(* AutoGeometry and AutoGroove-->Switch On/Off all Axis Power *)
	IF xToggleAllAxisPower THEN
		(* Step toggle Axis power *)
		CASE iStepAction OF
		(* check axis *)
		1:	IF NOT T_Station.TControl.xHardwareConfigError THEN
				xStepActionDone:=FALSE;
				iStepAction:=95;
				xTmp:=	T_Station.THardware.TAxisToolLeft.T_CtrleSingle.xDone
						AND T_Station.THardware.TAxisToolLeft.T_CtrleSingle.xNotMoving
						AND NOT(T_Station.THardware.TAxisToolLeft.T_CtrleSingle.xErr)
						AND NOT(T_Station.THardware.TAxisToolLeft.T_CtrleSingle.xExecute);
				xTmp:=	xTmp AND ((T_Station.THardware.TAxisToolCenter.T_CtrleSingle.xDone
						AND T_Station.THardware.TAxisToolCenter.T_CtrleSingle.xNotMoving
						AND NOT(T_Station.THardware.TAxisToolCenter.T_CtrleSingle.xErr)
						AND NOT(T_Station.THardware.TAxisToolCenter.T_CtrleSingle.xExecute) AND xMicroRodActive) OR NOT(xMicroRodActive)) ;
				xTmp:=	xTmp AND T_Station.THardware.TAxisToolRight.T_CtrleSingle.xDone
						AND T_Station.THardware.TAxisToolRight.T_CtrleSingle.xNotMoving
						AND NOT(T_Station.THardware.TAxisToolRight.T_CtrleSingle.xErr)
						AND NOT(T_Station.THardware.TAxisToolRight.T_CtrleSingle.xExecute);
				xTmp:=	xTmp AND T_Station.THardware.TAxisToolFeeder.T_CtrleSingle.xDone
						AND T_Station.THardware.TAxisToolFeeder.T_CtrleSingle.xNotMoving
						AND NOT(T_Station.THardware.TAxisToolFeeder.T_CtrleSingle.xErr)
						AND NOT(T_Station.THardware.TAxisToolFeeder.T_CtrleSingle.xExecute);
				xTmp:=	xTmp AND T_Station.THardware.TAxisGrindFeeder.T_CtrleSingle.xDone
						AND T_Station.THardware.TAxisGrindFeeder.T_CtrleSingle.xNotMoving
						AND NOT(T_Station.THardware.TAxisGrindFeeder.T_CtrleSingle.xErr)
						AND NOT(T_Station.THardware.TAxisGrindFeeder.T_CtrleSingle.xExecute);
				(* Start/Stop position or speed of teachin page has to be confirmed *)
				IF xTmp THEN
					iStepAction:=10;
				END_IF
			ELSE
				iStepAction:=95;
			END_IF;
		(* activ function axis *)
		10:	bStateMachine:=2;
			xSetStateMachine:=TRUE;
			xTmp:=	T_Station.THardware.TAxisToolLeft.T_CtrleSingle.xPower AND
					((T_Station.THardware.TAxisToolCenter.T_CtrleSingle.xPower AND xMicroRodActive) OR NOT(xMicroRodActive)) AND
					T_Station.THardware.TAxisToolRight.T_CtrleSingle.xPower AND
					T_Station.THardware.TAxisToolFeeder.T_CtrleSingle.xPower AND
					T_Station.THardware.TAxisGrindFeeder.T_CtrleSingle.xPower;
			IF xTmp THEN
				T_Station.THardware.TAxisToolLeft.T_CtrleSingle.iFunction:=4;
				IF xMicroRodActive THEN
					T_Station.THardware.TAxisToolCenter.T_CtrleSingle.iFunction:=4;
				END_IF;
				T_Station.THardware.TAxisToolRight.T_CtrleSingle.iFunction:=4;
				T_Station.THardware.TAxisToolFeeder.T_CtrleSingle.iFunction:=4;
				T_Station.THardware.TAxisGrindFeeder.T_CtrleSingle.iFunction:=4;
			ELSE
				IF NOT(T_Station.THardware.TAxisToolLeft.T_CtrleSingle.xPower) THEN
					T_Station.THardware.TAxisToolLeft.T_CtrleSingle.iFunction:=3;
				END_IF;
				IF xMicroRodActive THEN
					IF NOT(T_Station.THardware.TAxisToolCenter.T_CtrleSingle.xPower) THEN
						T_Station.THardware.TAxisToolCenter.T_CtrleSingle.iFunction:=3;
					END_IF;
				END_IF;
				IF NOT(T_Station.THardware.TAxisToolRight.T_CtrleSingle.xPower) THEN
					T_Station.THardware.TAxisToolRight.T_CtrleSingle.iFunction:=3;
				END_IF;
				IF NOT(T_Station.THardware.TAxisToolFeeder.T_CtrleSingle.xPower) THEN
					T_Station.THardware.TAxisToolFeeder.T_CtrleSingle.iFunction:=3;
				END_IF;
				IF NOT(T_Station.THardware.TAxisGrindFeeder.T_CtrleSingle.xPower) THEN
					T_Station.THardware.TAxisGrindFeeder.T_CtrleSingle.iFunction:=3;
				END_IF;
			END_IF;
			T_Station.THardware.TAxisToolLeft.T_CtrleSingle.xExecute:=TRUE;
			T_Station.THardware.TAxisToolCenter.T_CtrleSingle.xExecute:=xMicroRodActive;
			T_Station.THardware.TAxisToolRight.T_CtrleSingle.xExecute:=TRUE;
			T_Station.THardware.TAxisToolFeeder.T_CtrleSingle.xExecute:=TRUE;
			T_Station.THardware.TAxisGrindFeeder.T_CtrleSingle.xExecute:=TRUE;
			(* next step *)
			iStepAction:=20;
			xStepActionDone:=FALSE;
		(* confirm execution *)
		20:	IF NOT(xStepActionDone) THEN
			(* confirm execution *)
				T_Station.THardware.TAxisToolLeft.T_CtrleSingle.xExecute:=FALSE;
				T_Station.THardware.TAxisToolCenter.T_CtrleSingle.xExecute:=FALSE;
				T_Station.THardware.TAxisToolRight.T_CtrleSingle.xExecute:=FALSE;
				T_Station.THardware.TAxisToolFeeder.T_CtrleSingle.xExecute:=FALSE;
				T_Station.THardware.TAxisGrindFeeder.T_CtrleSingle.xExecute:=FALSE;
				xStepActionDone:=TRUE;
			ELSE
				xTmp:=	T_Station.THardware.TAxisToolLeft.T_CtrleSingle.xDone AND
						((T_Station.THardware.TAxisToolCenter.T_CtrleSingle.xDone AND xMicroRodActive) OR NOT(xMicroRodActive)) AND
						T_Station.THardware.TAxisToolRight.T_CtrleSingle.xDone AND
						T_Station.THardware.TAxisToolFeeder.T_CtrleSingle.xDone AND
						T_Station.THardware.TAxisGrindFeeder.T_CtrleSingle.xDone;
				IF xTmp THEN
				(* confirm action next step *)
					bStateMachine:=1;
					xSetStateMachine:=TRUE;
					iStepAction:=90;
					xStepActionDone:=FALSE;
				ELSE
					xTmp:=	T_Station.THardware.TAxisToolLeft.T_CtrleSingle.xErr OR
							(T_Station.THardware.TAxisToolCenter.T_CtrleSingle.xErr AND xMicroRodActive) OR
							T_Station.THardware.TAxisToolRight.T_CtrleSingle.xErr OR
							T_Station.THardware.TAxisToolFeeder.T_CtrleSingle.xErr OR
							T_Station.THardware.TAxisGrindFeeder.T_CtrleSingle.xErr;
					IF xTmp THEN
					(* activ action not ready or error *)
						iStepAction:=99;
						xStepActionDone:=FALSE;
					END_IF
				END_IF
			END_IF
		(* action done *)
		90:	T_Visu.ptrT_ExchgParam^.T_StationCommon.wState:=T_Visu.ptrT_ExchgParam^.T_StationCommon.wState AND 16#BF;
			T_Visu.T_CtrleAction.xDone:=TRUE;
			T_Visu.T_CtrleAction.xNotReady:=FALSE;
			T_Visu.T_CtrleAction.xErr:=FALSE;
			T_Visu.T_CtrleAction.udiErrorID:=0;
			xToggleAllAxisPower:=FALSE;
		(* axis not ready *)
		95:	T_Visu.ptrT_ExchgParam^.T_StationCommon.wState:=T_Visu.ptrT_ExchgParam^.T_StationCommon.wState AND 16#BF;
			TimerNotReady(IN:=TRUE);
			xToggleAllAxisPower:=FALSE;
		(* error *)
		99:	T_Visu.ptrT_ExchgParam^.T_StationCommon.wState:=T_Visu.ptrT_ExchgParam^.T_StationCommon.wState AND 16#BF;
			T_Visu.T_CtrleAction.xDone:=TRUE;
			T_Visu.T_CtrleAction.xNotReady:=FALSE;
			diErrorNr:=0;
			IF T_Station.THardware.TAxisToolLeft.T_CtrleSingle.xErr THEN
				diErrorNr:=1000000 + T_Station.THardware.TAxisToolLeft.T_CtrleSingle.udiErrorID;
			END_IF;
			IF xMicroRodActive THEN
				IF T_Station.THardware.TAxisToolCenter.T_CtrleSingle.xErr THEN
					diErrorNr:=2000000 + T_Station.THardware.TAxisToolCenter.T_CtrleSingle.udiErrorID;
				END_IF;
			END_IF;
			IF T_Station.THardware.TAxisToolRight.T_CtrleSingle.xErr THEN
				diErrorNr:=3000000 + T_Station.THardware.TAxisToolRight.T_CtrleSingle.udiErrorID;
			END_IF;
			IF T_Station.THardware.TAxisToolFeeder.T_CtrleSingle.xErr THEN
				diErrorNr:=4000000 + T_Station.THardware.TAxisToolFeeder.T_CtrleSingle.udiErrorID;
			END_IF;
			IF T_Station.THardware.TAxisGrindFeeder.T_CtrleSingle.xErr THEN
				diErrorNr:=5000000 + T_Station.THardware.TAxisGrindFeeder.T_CtrleSingle.udiErrorID;
			END_IF;
			FBErrorMessage(	diErrorNr:=diErrorNr,
							T_ErrorList:=T_ErrorList);
			T_Visu.ptrT_ExchgParam^.T_Visu.T_Message.sDynamicTextEnglish:=FBErrorMessage.sErrorTextEnglish;
			T_Visu.ptrT_ExchgParam^.T_Visu.T_Message.sDynamicTextDeutsch:=FBErrorMessage.sErrorTextDeutsch;
			T_Visu.ptrT_ExchgParam^.T_Visu.T_Message.sDynamicTextFrancais:=FBErrorMessage.sErrorTextFrancais;
			T_Visu.ptrT_ExchgParam^.T_SafetyCtrl.xSetForceError:=TRUE;
			T_Visu.ptrT_ExchgParam^.T_SafetyCtrl.diSetForceErrorNr:=diErrorNr;
			T_Visu.T_CtrleAction.xErr:=FALSE;
			T_Visu.T_CtrleAction.udiErrorID:=0;
			T_Station.THardware.TAxisToolLeft.T_CtrleSingle.iFunction:=1;
			T_Station.THardware.TAxisToolLeft.T_CtrleSingle.xExecute:=T_Station.THardware.TAxisToolLeft.T_CtrleSingle.xErr;
			IF xMicroRodActive THEN
				T_Station.THardware.TAxisToolCenter.T_CtrleSingle.iFunction:=1;
				T_Station.THardware.TAxisToolCenter.T_CtrleSingle.xExecute:=T_Station.THardware.TAxisToolCenter.T_CtrleSingle.xErr;
			END_IF;
			T_Station.THardware.TAxisToolRight.T_CtrleSingle.iFunction:=1;
			T_Station.THardware.TAxisToolRight.T_CtrleSingle.xExecute:=T_Station.THardware.TAxisToolRight.T_CtrleSingle.xErr;
			T_Station.THardware.TAxisToolFeeder.T_CtrleSingle.iFunction:=1;
			T_Station.THardware.TAxisToolFeeder.T_CtrleSingle.xExecute:=T_Station.THardware.TAxisToolFeeder.T_CtrleSingle.xErr;
			T_Station.THardware.TAxisGrindFeeder.T_CtrleSingle.iFunction:=1;
			T_Station.THardware.TAxisGrindFeeder.T_CtrleSingle.xExecute:=T_Station.THardware.TAxisGrindFeeder.T_CtrleSingle.xErr;
			xToggleAllAxisPower:=FALSE;
		END_CASE
	END_IF

(* Correction Tool Diameter +,++,-,-- *)
	IF xCorrectionToolDiameterAdd OR xCorrectionToolDiameterAddMore OR 	xCorrectionToolDiameterSub OR xCorrectionToolDiameterSubMore OR xResetToolDiameterCorrection OR xKeyPadActivation THEN
		CASE iStepAction OF
		(* check visu *)
		1:	xTmp:=	TRUE;
			IF xTmp THEN
				(* next Step *)
				iStepAction :=10;
				IF xResetToolDiameterCorrection THEN
					(* next Step *)
					iStepAction :=20;
				END_IF;
				IF xKeyPadActivation THEN
					IF (T_Visu.T_PlcParam.dwActualPage = 420) OR (T_Visu.T_PlcParam.dwActualPage = 11) OR (T_Visu.T_PlcParam.dwActualPage = 21) THEN
						(* next Step *)
						iStepAction :=30;
					END_IF;
					IF (T_Visu.T_PlcParam.dwActualPage = 430) THEN
						(* next Step *)
						iStepAction :=40;
					END_IF;
				END_IF;
			(* activ error *)
			ELSE iStepAction:=95; END_IF
		10:	IF xCorrectionToolDiameterAdd THEN
				rCorrectionValue:=0.1;
			END_IF;
			IF xCorrectionToolDiameterAddMore THEN
				rCorrectionValue:=1.0;
			END_IF;
			IF xCorrectionToolDiameterSub THEN
				rCorrectionValue:=-0.1;
			END_IF;
			IF xCorrectionToolDiameterSubMore THEN
				rCorrectionValue:=-1.0;
			END_IF;
			T_Visu.ptrT_ExchgParam^.T_InfoValueCommon.rCorrectionToolDiameter:=T_Visu.ptrT_ExchgParam^.T_InfoValueCommon.rCorrectionToolDiameter + rCorrectionValue;
			IF (T_Visu.ptrT_ExchgParam^.T_InfoValueCommon.rCorrectionToolDiameter < 0.1) AND
			    (T_Visu.ptrT_ExchgParam^.T_InfoValueCommon.rCorrectionToolDiameter > -0.1) THEN
				T_Visu.ptrT_ExchgParam^.T_InfoValueCommon.rCorrectionToolDiameter:=0.0;
			END_IF;
			(* next Step *)
			iStepAction :=90;
		20:	T_Visu.ptrT_ExchgParam^.T_InfoValueCommon.rCorrectionToolDiameter:=0.0;
			(* next Step *)
			iStepAction :=90;
		30:	T_Visu.ptrT_ExchgParam^.T_InfoValueCommon.xKeyPadActivation:=NOT(T_Visu.ptrT_ExchgParam^.T_InfoValueCommon.xKeyPadActivation);
			(* next Step *)
			iStepAction :=90;
		40:	(* 0= 3 value prisma, 1 = 3 value prisma input para, 2 = 2 value prisma, 3 = 2 value prisma input para *)
			IF (T_Visu.ptrT_ExchgParam^.T_StationCommon.T_PrismPara.bStateInputPrisma = 0) THEN
				T_Visu.ptrT_ExchgParam^.T_StationCommon.T_PrismPara.bStateInputPrisma:=1;
			ELSIF (T_Visu.ptrT_ExchgParam^.T_StationCommon.T_PrismPara.bStateInputPrisma = 1) THEN
				T_Visu.ptrT_ExchgParam^.T_StationCommon.T_PrismPara.bStateInputPrisma:=0;
			ELSIF (T_Visu.ptrT_ExchgParam^.T_StationCommon.T_PrismPara.bStateInputPrisma = 2) THEN
				T_Visu.ptrT_ExchgParam^.T_StationCommon.T_PrismPara.bStateInputPrisma:=3;
			ELSIF (T_Visu.ptrT_ExchgParam^.T_StationCommon.T_PrismPara.bStateInputPrisma = 3) THEN
				T_Visu.ptrT_ExchgParam^.T_StationCommon.T_PrismPara.bStateInputPrisma:=2;
			END_IF;
			(* next Step *)
			iStepAction:=90;
		(* change page done *)
		90:	T_Visu.T_CtrleAction.xDone:=TRUE;
			T_Visu.T_CtrleAction.xNotReady:=FALSE;
			T_Visu.T_CtrleAction.xErr:=FALSE;
			T_Visu.T_CtrleAction.udiErrorID:=0;
			xCorrectionToolDiameterAdd:=xCorrectionToolDiameterAddMore:=xCorrectionToolDiameterSub:=xCorrectionToolDiameterSubMore:=xResetToolDiameterCorrection:=xKeyPadActivation:=FALSE;
		(* not ready *)
		95:	T_Visu.T_CtrleAction.xDone:=TRUE;
			T_Visu.T_CtrleAction.xNotReady:=FALSE;
			T_Visu.T_CtrleAction.xErr:=FALSE;
			T_Visu.T_CtrleAction.udiErrorID:=0;
			xCorrectionToolDiameterAdd:=xCorrectionToolDiameterAddMore:=xCorrectionToolDiameterSub:=xCorrectionToolDiameterSubMore:=xResetToolDiameterCorrection:=xKeyPadActivation:=FALSE;
		END_CASE
	END_IF;

(* Function Correction Tool Diameter *)
	IF xFctCorrectionToolDiameter THEN
		CASE iStepAction OF
		(* check axis *)
		1:	IF NOT T_Station.TControl.xHardwareConfigError THEN
				xStepActionDone:=FALSE;
				iStepAction:=95;
				xTmp:=	T_Station.THardware.TAxisGrindFeeder.T_CtrleSingle.xDone
						AND T_Station.THardware.TAxisGrindFeeder.T_CtrleSingle.xReady
						AND T_Station.THardware.TAxisGrindFeeder.T_CtrleSingle.xNotMoving
						AND NOT(T_Station.THardware.TAxisGrindFeeder.T_CtrleSingle.xErr)
						AND NOT(T_Station.THardware.TAxisGrindFeeder.T_CtrleSingle.xExecute);
				(* Start/Stop position or speed of teachin page has to be confirmed *)
				IF xTmp THEN
					iStepAction:=10;
				END_IF
			ELSE
				iStepAction:=95;
			END_IF;
		(* Display message to ask for confirmation *)
		10:	T_Visu.ptrT_ExchgParam^.T_Visu.T_Message.iState:=108;
			iStepAction:=20;
		(* waiting for key <Enter> or <Esc> *)
		20:	IF RisingEdgeKeyPanel_Enter.Q THEN iStepAction:=30;
			ELSE IF RisingEdgeKeyPanel_Esc.Q THEN iStepAction:=90; END_IF END_IF
			(* An other message has been displayed, stop teach action *)
			IF T_Visu.ptrT_ExchgParam^.T_Visu.T_Message.iState<>108 THEN iStepAction:=90; END_IF
		(* activ function axis *)
		30:	(*T_Visu.ptrT_ExchgParam^.T_InfoValueCommon.rActualGrindAxisPosition:=T_Visu.ptrT_ExchgParam^.T_InfoValueCommon.rActualGrindAxisPosition - T_Visu.ptrT_ExchgParam^.T_InfoValueCommon.rCorrectionToolDiameter;*)
			T_Station.THardware.TAxisGrindFeeder.T_CtrleSingle.rSetPosition:=T_Station.THardware.TAxisGrindFeeder.T_LiveValue.lrActualPosition - T_Visu.ptrT_ExchgParam^.T_InfoValueCommon.rCorrectionToolDiameter;
			T_Visu.ptrT_ExchgParam^.T_InfoValueCommon.rCorrectionToolDiameter:=0.0;
			T_Station.THardware.TAxisGrindFeeder.T_CtrleSingle.iFunction:=11;
			T_Station.THardware.TAxisGrindFeeder.T_CtrleSingle.xExecute:=TRUE;
			(* next step *)
			iStepAction:=50;
			xStepActionDone:=FALSE;
		(* confirm execution *)
		50:	IF NOT(xStepActionDone) THEN
			(* confirm execution *)
				T_Station.THardware.TAxisGrindFeeder.T_CtrleSingle.xExecute:=FALSE;
				xStepActionDone:=TRUE;
			ELSE
				IF T_Station.THardware.TAxisGrindFeeder.T_CtrleSingle.xDone THEN
				(* confirm action next step *)
					iStepAction:=90;
					xStepActionDone:=FALSE;
				ELSE
					IF T_Station.THardware.TAxisGrindFeeder.T_CtrleSingle.xErr THEN
					(* activ action not ready or error *)
						iStepAction:=99;
						xStepActionDone:=FALSE;
					END_IF
				END_IF
			END_IF
		(* action done *)
		90:	T_Visu.ptrT_ExchgParam^.T_StationCommon.wState:=T_Visu.ptrT_ExchgParam^.T_StationCommon.wState AND 16#BF;
			T_Visu.T_CtrleAction.xDone:=TRUE;
			T_Visu.T_CtrleAction.xNotReady:=FALSE;
			T_Visu.T_CtrleAction.xErr:=FALSE;
			T_Visu.T_CtrleAction.udiErrorID:=0;
			xFctCorrectionToolDiameter:=FALSE;
		(* axis not ready *)
		95:	T_Visu.ptrT_ExchgParam^.T_StationCommon.wState:=T_Visu.ptrT_ExchgParam^.T_StationCommon.wState AND 16#BF;
			TimerNotReady(IN:=TRUE);
			xFctCorrectionToolDiameter:=FALSE;
		(* error *)
		99:	T_Visu.ptrT_ExchgParam^.T_StationCommon.wState:=T_Visu.ptrT_ExchgParam^.T_StationCommon.wState AND 16#BF;
			T_Visu.T_CtrleAction.xDone:=TRUE;
			T_Visu.T_CtrleAction.xNotReady:=FALSE;
			IF (T_Station.THardware.TAxisGrindFeeder.T_Config_Gen.iTyp <> 0) THEN
				diErrorNr:=(T_Station.THardware.TAxisGrindFeeder.T_Config_Gen.iTyp * 1000000) + T_Station.THardware.TAxisGrindFeeder.T_CtrleSingle.udiErrorID;
			ELSE
				diErrorNr:=0;
			END_IF;
			FBErrorMessage(	diErrorNr:=diErrorNr,
							T_ErrorList:=T_ErrorList);
			T_Visu.ptrT_ExchgParam^.T_Visu.T_Message.sDynamicTextEnglish:=FBErrorMessage.sErrorTextEnglish;
			T_Visu.ptrT_ExchgParam^.T_Visu.T_Message.sDynamicTextDeutsch:=FBErrorMessage.sErrorTextDeutsch;
			T_Visu.ptrT_ExchgParam^.T_Visu.T_Message.sDynamicTextFrancais:=FBErrorMessage.sErrorTextFrancais;
			T_Visu.ptrT_ExchgParam^.T_SafetyCtrl.xSetForceError:=TRUE;
			T_Visu.ptrT_ExchgParam^.T_SafetyCtrl.diSetForceErrorNr:=diErrorNr;
			T_Visu.T_CtrleAction.xErr:=FALSE;
			T_Visu.T_CtrleAction.udiErrorID:=0;
			T_Station.THardware.TAxisGrindFeeder.T_CtrleSingle.iFunction:=1;
			T_Station.THardware.TAxisGrindFeeder.T_CtrleSingle.xExecute:=TRUE;
			xFctCorrectionToolDiameter:=FALSE;
		END_CASE
	END_IF;

(* Select Prisma 1 or 2 Input *)
	IF xSelectPrisma THEN
		CASE iStepAction OF
		(* check visu *)
		1:	xTmp:=	TRUE;
			IF xTmp THEN
				(* next Step *)
				iStepAction :=10;
			(* activ error *)
			ELSE iStepAction:=95; END_IF
		10:	(* 0= 3 value prisma, 1 = 3 value prisma input para, 2 = 2 value prisma, 3 = 2 value prisma input para *)
			IF (T_Visu.ptrT_ExchgParam^.T_StationCommon.T_PrismPara.bStateInputPrisma = 0) OR (T_Visu.ptrT_ExchgParam^.T_StationCommon.T_PrismPara.bStateInputPrisma = 1) THEN
				T_Visu.ptrT_ExchgParam^.T_StationCommon.T_PrismPara.bStateInputPrisma:=2;
			ELSIF (T_Visu.ptrT_ExchgParam^.T_StationCommon.T_PrismPara.bStateInputPrisma = 2) OR (T_Visu.ptrT_ExchgParam^.T_StationCommon.T_PrismPara.bStateInputPrisma = 3) THEN
				T_Visu.ptrT_ExchgParam^.T_StationCommon.T_PrismPara.bStateInputPrisma:=0;
			END_IF;
			(* next Step *)
			iStepAction:=90;
		(* change page done *)
		90:	T_Visu.T_CtrleAction.xDone:=TRUE;
			T_Visu.T_CtrleAction.xNotReady:=FALSE;
			T_Visu.T_CtrleAction.xErr:=FALSE;
			T_Visu.T_CtrleAction.udiErrorID:=0;
			xSelectPrisma:=FALSE;
		(* not ready *)
		95:	T_Visu.T_CtrleAction.xDone:=TRUE;
			T_Visu.T_CtrleAction.xNotReady:=FALSE;
			T_Visu.T_CtrleAction.xErr:=FALSE;
			T_Visu.T_CtrleAction.udiErrorID:=0;
			xSelectPrisma:=FALSE;
		END_CASE
	END_IF;

(* Set calculated ToolRotation Torque *)
	IF xSetCalculToolRotTorque THEN
		CASE iStepAction OF
		(* check visu *)
		1:	xTmp:=	TRUE;
			IF xTmp THEN
				(* next Step *)
				iStepAction :=10;
			(* activ error *)
			ELSE iStepAction:=95; END_IF
		10:	uiToolLeftZeroTorque:=T_Station.THardware.TAxisToolLeft.T_LiveValue.uiActualTorque;
			FBCalcTorqueToolLeft(	xStart:=TRUE,
									uiActualTorque:= T_Station.THardware.TAxisToolLeft.T_LiveValue.uiActualTorque,
									uiZeroTorque:=uiToolLeftZeroTorque,
									iStepCalc:= 100);
			uiToolCenterZeroTorque:=T_Station.THardware.TAxisToolCenter.T_LiveValue.uiActualTorque;
			FBCalcTorqueToolCenter(	xStart:=TRUE,
									uiActualTorque:= T_Station.THardware.TAxisToolCenter.T_LiveValue.uiActualTorque,
									uiZeroTorque:=uiToolCenterZeroTorque,
									iStepCalc:= 100);
			uiToolRightZeroTorque:=T_Station.THardware.TAxisToolRight.T_LiveValue.uiActualTorque;
			FBCalcTorqueToolRight(	xStart:=TRUE,
									uiActualTorque:= T_Station.THardware.TAxisToolRight.T_LiveValue.uiActualTorque,
									uiZeroTorque:=uiToolRightZeroTorque,
									iStepCalc:= 100);
			(* next Step *)
			iStepAction:=90;
		(* change page done *)
		90:	T_Visu.T_CtrleAction.xDone:=TRUE;
			T_Visu.T_CtrleAction.xNotReady:=FALSE;
			T_Visu.T_CtrleAction.xErr:=FALSE;
			T_Visu.T_CtrleAction.udiErrorID:=0;
			xSetCalculToolRotTorque:=FALSE;
		(* not ready *)
		95:	T_Visu.T_CtrleAction.xDone:=TRUE;
			T_Visu.T_CtrleAction.xNotReady:=FALSE;
			T_Visu.T_CtrleAction.xErr:=FALSE;
			T_Visu.T_CtrleAction.udiErrorID:=0;
			xSetCalculToolRotTorque:=FALSE;
		END_CASE
	END_IF;

(* Reset calculated ToolRotation Torque *)
	IF xResetCalculToolRotTorque THEN
		CASE iStepAction OF
		(* check visu *)
		1:	xTmp:=	TRUE;
			IF xTmp THEN
				(* next Step *)
				iStepAction :=10;
			(* activ error *)
			ELSE iStepAction:=95; END_IF
		10:	uiToolLeftZeroTorque:=0;
			FBCalcTorqueToolLeft(	xStart:=TRUE,
									uiActualTorque:= T_Station.THardware.TAxisToolLeft.T_LiveValue.uiActualTorque,
									uiZeroTorque:=uiToolLeftZeroTorque,
									iStepCalc:= 100);
			uiToolCenterZeroTorque:=0;
			FBCalcTorqueToolCenter(	xStart:=TRUE,
									uiActualTorque:= T_Station.THardware.TAxisToolCenter.T_LiveValue.uiActualTorque,
									uiZeroTorque:=uiToolCenterZeroTorque,
									iStepCalc:= 100);
			uiToolRightZeroTorque:=0;
			FBCalcTorqueToolRight(	xStart:=TRUE,
									uiActualTorque:= T_Station.THardware.TAxisToolRight.T_LiveValue.uiActualTorque,
									uiZeroTorque:=uiToolRightZeroTorque,
									iStepCalc:= 100);
			(* next Step *)
			iStepAction:=90;
		(* change page done *)
		90:	T_Visu.T_CtrleAction.xDone:=TRUE;
			T_Visu.T_CtrleAction.xNotReady:=FALSE;
			T_Visu.T_CtrleAction.xErr:=FALSE;
			T_Visu.T_CtrleAction.udiErrorID:=0;
			xResetCalculToolRotTorque:=FALSE;
		(* not ready *)
		95:	T_Visu.T_CtrleAction.xDone:=TRUE;
			T_Visu.T_CtrleAction.xNotReady:=FALSE;
			T_Visu.T_CtrleAction.xErr:=FALSE;
			T_Visu.T_CtrleAction.udiErrorID:=0;
			xResetCalculToolRotTorque:=FALSE;
		END_CASE
	END_IF;

(* Switch WireFeed Jog Speed Slow/Fast *)
	IF xSlowFastJogToolRotation OR xSlowFastJogToolFeeder OR xSlowFastJogGrindFeeder THEN
		CASE iStepAction OF
		(* check visu *)
		1:	xTmp:=	TRUE;
			IF xTmp THEN
				(* next Step *)
				iStepAction :=10;
			(* activ error *)
			ELSE iStepAction:=95; END_IF
		10:	IF xSlowFastJogToolRotation THEN
				T_Visu.ptrT_ExchgParam^.T_TeachIn.xSlowFastToolRotation:=NOT(T_Visu.ptrT_ExchgParam^.T_TeachIn.xSlowFastToolRotation);
			END_IF;
			IF xSlowFastJogToolFeeder THEN
				T_Visu.ptrT_ExchgParam^.T_TeachIn.xSlowFastToolFeed:=NOT(T_Visu.ptrT_ExchgParam^.T_TeachIn.xSlowFastToolFeed);
			END_IF;
			IF xSlowFastJogGrindFeeder THEN
				T_Visu.ptrT_ExchgParam^.T_TeachIn.xSlowFastGrindFeeder:=NOT(T_Visu.ptrT_ExchgParam^.T_TeachIn.xSlowFastGrindFeeder);
			END_IF;
			(* next Step *)
			iStepAction:=90;
		(* change page done *)
		90:	T_Visu.T_CtrleAction.xDone:=TRUE;
			T_Visu.T_CtrleAction.xNotReady:=FALSE;
			T_Visu.T_CtrleAction.xErr:=FALSE;
			T_Visu.T_CtrleAction.udiErrorID:=0;
			xSlowFastJogToolRotation:=xSlowFastJogToolFeeder:=xSlowFastJogGrindFeeder:=FALSE;
		(* not ready *)
		95:	T_Visu.T_CtrleAction.xDone:=TRUE;
			T_Visu.T_CtrleAction.xNotReady:=FALSE;
			T_Visu.T_CtrleAction.xErr:=FALSE;
			T_Visu.T_CtrleAction.udiErrorID:=0;
			xSlowFastJogToolRotation:=xSlowFastJogToolFeeder:=xSlowFastJogGrindFeeder:=FALSE;
		END_CASE
	END_IF;

(* Action stop axis *)
	IF xStopAxis THEN
		(* Step stop axis *)
		CASE iStepAction OF
		(* check axis *)
		1:	xMoveAbsPosition:=xMoveRelPosition:=xMoveContinousVel:=FALSE;
			IF NOT T_Station.TControl.xHardwareConfigError THEN
				xStepActionDone:=FALSE;
				IF ptrTeachINAxis^.T_CtrleSingle.xErr THEN
					iStepAction:=99;
					RETURN;
				END_IF;
				iStepAction:=95;
				xTmp:=	ptrTeachINAxis^.T_CtrleSingle.xReady (*AND
						NOT(ptrTeachINAxis^.T_CtrleSingle.xErr)*);
				(* Start/Stop position or speed of teachin page has to be confirmed *)
				IF xTmp THEN
					iStepAction:=10;
				ELSE
					iStepAction:=95;
				END_IF
			ELSE
				iStepAction:=95;
			END_IF;
		(* activ function axis *)
		10:	ptrTeachINAxis^.T_CtrleSingle.iFunction:=5;
			ptrTeachINAxis^.T_CtrleSingle.xExecute:=TRUE;
			(* init. acc/dec/jerk *)
			ptrTeachINAxis^.T_CtrleSingle.lrAcceleration:=TParaAxisTeachIN.rAcceleration;
			ptrTeachINAxis^.T_CtrleSingle.lrDecceleration:=TParaAxisTeachIN.rDeceleration;
			(*
			ptrTeachINAxis^.T_CtrleSingle.lrAcceleration:=ptrTeachINAxis^.T_Config_ObjFileValue.lrAcceleration;
			ptrTeachINAxis^.T_CtrleSingle.lrDecceleration:=ptrTeachINAxis^.T_Config_ObjFileValue.lrDecceleration;
			ptrTeachINAxis^.T_CtrleSingle.lrJerk:=ptrTeachINAxis^.T_Config_ObjFileValue.lrJerk;
			*)
			(* next step *)
			iStepAction:=20;
			xStepActionDone:=FALSE;
		(* waiting stop confirmation *)
		20:	IF NOT(xStepActionDone) THEN
			(* confirm execution *)
				ptrTeachINAxis^.T_CtrleSingle.xExecute:=FALSE;
				xStepActionDone:=TRUE;
			ELSE
				IF ptrTeachINAxis^.T_CtrleSingle.xDone THEN
				(* confirm action next step *)
					iStepAction:=90;
					xStepActionDone:=FALSE;
				ELSE
					IF ptrTeachINAxis^.T_CtrleSingle.xErr THEN
					(* activ action not ready or error *)
						iStepAction:=99;
						xStepActionDone:=FALSE;
					END_IF
				END_IF
			END_IF
		(* waiting time out *)
		89:	IF TimerAction.Q THEN iStepAction:=90; END_IF
			(*T_Visu.ptrT_ExchgParam^.T_TeachIn.iStateAxisMovement:=1;*)
		(* action done *)
		90:	bStateMachine:=1;
			xSetStateMachine:=TRUE;
			T_Visu.ptrT_ExchgParam^.T_StationCommon.wState:=T_Visu.ptrT_ExchgParam^.T_StationCommon.wState AND 16#BF;
			T_Visu.T_CtrleAction.xDone:=TRUE;
			T_Visu.T_CtrleAction.xNotReady:=FALSE;
			T_Visu.T_CtrleAction.xErr:=FALSE;
			T_Visu.T_CtrleAction.udiErrorID:=0;
			xStopAxis:=FALSE;
			(*T_Visu.ptrT_ExchgParam^.T_TeachIn.iStateAxisMovement:=1;*)
		(* axis not ready *)
		95:	T_Visu.ptrT_ExchgParam^.T_StationCommon.wState:=T_Visu.ptrT_ExchgParam^.T_StationCommon.wState AND 16#BF;
			TimerNotReady(IN:=TRUE);
			xStopAxis:=FALSE;
			(*T_Visu.ptrT_ExchgParam^.T_TeachIn.iStateAxisMovement:=1;*)
		(* error *)
		99:	T_Visu.ptrT_ExchgParam^.T_StationCommon.wState:=T_Visu.ptrT_ExchgParam^.T_StationCommon.wState AND 16#BF;
			T_Visu.T_CtrleAction.xDone:=TRUE;
			T_Visu.T_CtrleAction.xNotReady:=FALSE;
			IF (ptrTeachINAxis^.T_Config_Gen.iTyp <> 0) THEN
				diErrorNr:=(ptrTeachINAxis^.T_Config_Gen.iTyp * 1000000) + ptrTeachINAxis^.T_CtrleSingle.udiErrorID;
			ELSE
				diErrorNr:=0;
			END_IF;
			FBErrorMessage(	diErrorNr:=diErrorNr,
							T_ErrorList:=T_ErrorList);
			T_Visu.ptrT_ExchgParam^.T_Visu.T_Message.sDynamicTextEnglish:=FBErrorMessage.sErrorTextEnglish;
			T_Visu.ptrT_ExchgParam^.T_Visu.T_Message.sDynamicTextDeutsch:=FBErrorMessage.sErrorTextDeutsch;
			T_Visu.ptrT_ExchgParam^.T_Visu.T_Message.sDynamicTextFrancais:=FBErrorMessage.sErrorTextFrancais;
			T_Visu.ptrT_ExchgParam^.T_SafetyCtrl.xSetForceError:=TRUE;
			T_Visu.ptrT_ExchgParam^.T_SafetyCtrl.diSetForceErrorNr:=diErrorNr;
			T_Visu.T_CtrleAction.xErr:=FALSE;
			T_Visu.T_CtrleAction.udiErrorID:=0;
			ptrTeachINAxis^.T_CtrleSingle.iFunction:=1;
			ptrTeachINAxis^.T_CtrleSingle.xExecute:=TRUE;
			xStopAxis:=FALSE;
			T_StartUp.T_Ctrle.xSetSecurityStateON:=TRUE;
		END_CASE
	END_IF

(* Action move abs position *)
	IF xMoveAbsPosition OR xMoveRelPosition THEN
		(* Step move abs position *)
		CASE iStepAction OF
		(* check axis *)
		1:	IF NOT T_Station.TControl.xHardwareConfigError THEN
				xStepActionDone:=FALSE;
				iStepAction:=95;
				xTmp:=	ptrTeachINAxis^.T_CtrleSingle.xDone
						AND ptrTeachINAxis^.T_CtrleSingle.xReady
						AND ptrTeachINAxis^.T_CtrleSingle.xNotMoving
						AND ptrTeachINAxis^.T_CtrleSingle.xPower
						AND NOT(ptrTeachINAxis^.T_CtrleSingle.xErr)
						AND NOT(ptrTeachINAxis^.T_CtrleSingle.xExecute)
(*24.09.2010: KFS	{	 *)
						AND( (  T_Visu.T_PlcParam.dwActualPage = 210
							   AND NOT(T_Station.THardware.TCylToolLeftActive.T_CtrleCyl.T_Standard.xActivOn)
							   AND NOT(T_Station.THardware.TCylToolRightActive.T_CtrleCyl.T_Standard.xActivOn)
					     		   AND NOT(T_Station.THardware.TCylToolCenterActive.T_CtrleCyl.T_Standard.xActivOn) )  OR ( T_Visu.T_PlcParam.dwActualPage <> 210))
(*24.09.2010: KFS	}	 *)
						AND ((ptrTeachINAxis^.T_CtrleSingle.xRef AND xMoveAbsPosition AND xMicroRodActive) OR NOT(xMicroRodActive)OR xMoveRelPosition);
				(* Start/Stop position or speed of teachin page has to be confirmed *)
				IF xTmp THEN
					iStepAction:=10;
				ELSE
					IF NOT ptrTeachINAxis^.T_CtrleSingle.xRef AND xMoveAbsPosition THEN
					(* Display message, axis not referenced *)
						tTimeOutAction:=TimerAction.ET+T#2s;
						T_Visu.ptrT_ExchgParam^.T_Visu.T_Message.iState:=18;
						(* Action has been cancelled *)
						iStepAction:=89;
					END_IF
				END_IF
			ELSE
				iStepAction:=95;
			END_IF;
		(* activ function axis *)
		10:	tTimeOutAction:=T#999s;
			bStateMachine:=2;
			xSetStateMachine:=TRUE;
			IF xMoveAbsPosition THEN iStepAction:=20; END_IF
			IF xMoveRelPosition THEN iStepAction:=35; END_IF
			(* init. acc/dec/jerk *)
			ptrTeachINAxis^.T_CtrleSingle.lrAcceleration:=TParaAxisTeachIN.rAcceleration;
			ptrTeachINAxis^.T_CtrleSingle.lrDecceleration:=TParaAxisTeachIN.rDeceleration;
			(*
			ptrTeachINAxis^.T_CtrleSingle.lrAcceleration:=ptrTeachINAxis^.T_Config_ObjFileValue.lrAcceleration;
			ptrTeachINAxis^.T_CtrleSingle.lrDecceleration:=ptrTeachINAxis^.T_Config_ObjFileValue.lrDecceleration;
			ptrTeachINAxis^.T_CtrleSingle.lrJerk:=ptrTeachINAxis^.T_Config_ObjFileValue.lrJerk;
			*)
		(* activ function axis move absolut *)
		20:	ptrTeachINAxis^.T_CtrleSingle.iFunction:=7;
			ptrTeachINAxis^.T_CtrleSingle.xExecute:=TRUE;
			(* next step *)
			iStepAction:=40;
			xStepActionDone:=FALSE;
		(* activ function axis move relativ *)
		35:	ptrTeachINAxis^.T_CtrleSingle.iFunction:=8;
			ptrTeachINAxis^.T_CtrleSingle.xExecute:=TRUE;
			(* next step *)
			iStepAction:=40;
			xStepActionDone:=FALSE;
		(* confirm execution *)
		40:	IF NOT(xStepActionDone) THEN
			(* confirm execution *)
				ptrTeachINAxis^.T_CtrleSingle.xExecute:=FALSE;
				xStepActionDone:=TRUE;
				(* Display message, 'Start moving' *)
				T_Visu.ptrT_ExchgParam^.T_Visu.T_Message.iState:=26;
			ELSE
				IF ptrTeachINAxis^.T_CtrleSingle.xDone THEN
				(* confirm action next step *)
					bStateMachine:=1;
					xSetStateMachine:=TRUE;
					iStepAction:=90;
					xStepActionDone:=FALSE;
				ELSE
					IF ptrTeachINAxis^.T_CtrleSingle.xErr THEN
					(* activ action not ready or error *)
						iStepAction:=99;
						xStepActionDone:=FALSE;
					END_IF
				END_IF
			END_IF
		(* waiting timeout *)
		89: IF TimerAction.Q THEN iStepAction:=90; END_IF
			(*T_Visu.ptrT_ExchgParam^.T_TeachIn.iStateAxisMovement:=1;*)
		(* action done *)
		90:	T_Visu.ptrT_ExchgParam^.T_StationCommon.wState:=T_Visu.ptrT_ExchgParam^.T_StationCommon.wState AND 16#BF;
			T_Visu.T_CtrleAction.xDone:=TRUE;
			T_Visu.T_CtrleAction.xNotReady:=FALSE;
			T_Visu.T_CtrleAction.xErr:=FALSE;
			T_Visu.T_CtrleAction.udiErrorID:=0;
			xMoveAbsPosition:=FALSE;
			xMoveRelPosition:=FALSE;
			(*T_Visu.ptrT_ExchgParam^.T_TeachIn.iStateAxisMovement:=1;*)
		(* axis not ready *)
		95:	T_Visu.ptrT_ExchgParam^.T_StationCommon.wState:=T_Visu.ptrT_ExchgParam^.T_StationCommon.wState AND 16#BF;
			TimerNotReady(IN:=TRUE);
			xMoveAbsPosition:=FALSE;
			xMoveRelPosition:=FALSE;
			(*T_Visu.ptrT_ExchgParam^.T_TeachIn.iStateAxisMovement:=1;*)
		(* error *)
		99:	T_Visu.ptrT_ExchgParam^.T_StationCommon.wState:=T_Visu.ptrT_ExchgParam^.T_StationCommon.wState AND 16#BF;
			T_Visu.T_CtrleAction.xDone:=TRUE;
			T_Visu.T_CtrleAction.xNotReady:=FALSE;
			IF (ptrTeachINAxis^.T_Config_Gen.iTyp <> 0) THEN
				diErrorNr:=(ptrTeachINAxis^.T_Config_Gen.iTyp * 1000000) + ptrTeachINAxis^.T_CtrleSingle.udiErrorID;
			ELSE
				diErrorNr:=0;
			END_IF;
			FBErrorMessage(	diErrorNr:=diErrorNr,
							T_ErrorList:=T_ErrorList);
			T_Visu.ptrT_ExchgParam^.T_Visu.T_Message.sDynamicTextEnglish:=FBErrorMessage.sErrorTextEnglish;
			T_Visu.ptrT_ExchgParam^.T_Visu.T_Message.sDynamicTextDeutsch:=FBErrorMessage.sErrorTextDeutsch;
			T_Visu.ptrT_ExchgParam^.T_Visu.T_Message.sDynamicTextFrancais:=FBErrorMessage.sErrorTextFrancais;
			T_Visu.ptrT_ExchgParam^.T_SafetyCtrl.xSetForceError:=TRUE;
			T_Visu.ptrT_ExchgParam^.T_SafetyCtrl.diSetForceErrorNr:=diErrorNr;
			T_Visu.T_CtrleAction.xErr:=FALSE;
			T_Visu.T_CtrleAction.udiErrorID:=0;
			ptrTeachINAxis^.T_CtrleSingle.iFunction:=1;
			ptrTeachINAxis^.T_CtrleSingle.xExecute:=TRUE;
			xMoveAbsPosition:=FALSE;
			xMoveRelPosition:=FALSE;
			T_StartUp.T_Ctrle.xSetSecurityStateON:=TRUE;
			(*T_Visu.ptrT_ExchgParam^.T_TeachIn.iStateAxisMovement:=1;*)
		END_CASE
	END_IF

(* Action move velocity *)
	IF xMoveContinousVel THEN
		(* Step move continuous velocity *)
		CASE iStepAction OF
		(* check axis *)
		1:	IF NOT T_Station.TControl.xHardwareConfigError THEN
				xStepActionDone:=FALSE;
				iStepAction:=95;
				xTmp:=	ptrTeachINAxis^.T_CtrleSingle.xDone
						AND ptrTeachINAxis^.T_CtrleSingle.xReady
						AND ptrTeachINAxis^.T_CtrleSingle.xNotMoving
						AND ptrTeachINAxis^.T_CtrleSingle.xPower
						AND NOT(ptrTeachINAxis^.T_CtrleSingle.xErr)
						AND NOT(ptrTeachINAxis^.T_CtrleSingle.xExecute)
(*24.09.2010: KFS	{	 *)
						AND( (  T_Visu.T_PlcParam.dwActualPage = 210
							   AND NOT(T_Station.THardware.TCylToolLeftActive.T_CtrleCyl.T_Standard.xActivOn)
							   AND NOT(T_Station.THardware.TCylToolRightActive.T_CtrleCyl.T_Standard.xActivOn)
					     		   AND NOT(T_Station.THardware.TCylToolCenterActive.T_CtrleCyl.T_Standard.xActivOn) )  OR ( T_Visu.T_PlcParam.dwActualPage <> 210))
(*24.09.2010: KFS	}	 *)
						AND (ptrTeachINAxis^.T_CtrleSingle.lrVelocity <> 0);
				(* Start/Stop position or speed of teachin page has to be confirmed *)
				IF xTmp THEN
					iStepAction:=10;
				END_IF
			ELSE
				iStepAction:=95;
			END_IF;
		(* activ function axis *)
		10:	bStateMachine:=2;
			xSetStateMachine:=TRUE;
			ptrTeachINAxis^.T_CtrleSingle.iFunction:=6;
			ptrTeachINAxis^.T_CtrleSingle.xExecute:=TRUE;
			(* init. acc/dec/jerk *)
			ptrTeachINAxis^.T_CtrleSingle.lrAcceleration:=TParaAxisTeachIN.rAcceleration;
			ptrTeachINAxis^.T_CtrleSingle.lrDecceleration:=TParaAxisTeachIN.rDeceleration;
			(*
			ptrTeachINAxis^.T_CtrleSingle.lrAcceleration:=ptrTeachINAxis^.T_Config_ObjFileValue.lrAcceleration;
			ptrTeachINAxis^.T_CtrleSingle.lrDecceleration:=ptrTeachINAxis^.T_Config_ObjFileValue.lrDecceleration;
			ptrTeachINAxis^.T_CtrleSingle.lrJerk:=ptrTeachINAxis^.T_Config_ObjFileValue.lrJerk;
			*)
			(* next step *)
			iStepAction:=20;
			xStepActionDone:=FALSE;
		(* confirm execution *)
		20:	IF NOT(xStepActionDone) THEN
			(* confirm execution *)
				ptrTeachINAxis^.T_CtrleSingle.xExecute:=FALSE;
				xStepActionDone:=TRUE;
			ELSE
				IF ptrTeachINAxis^.T_CtrleSingle.xDone THEN
				(* confirm action next step *)
					iStepAction:=90;
					xStepActionDone:=FALSE;
				ELSE
					IF ptrTeachINAxis^.T_CtrleSingle.xErr THEN
					(* activ action not ready or error *)
						iStepAction:=99;
						xStepActionDone:=FALSE;
					END_IF
				END_IF
			END_IF
		(* action done *)
		90:	T_Visu.ptrT_ExchgParam^.T_StationCommon.wState:=T_Visu.ptrT_ExchgParam^.T_StationCommon.wState AND 16#BF;
			T_Visu.T_CtrleAction.xDone:=TRUE;
			T_Visu.T_CtrleAction.xNotReady:=FALSE;
			T_Visu.T_CtrleAction.xErr:=FALSE;
			T_Visu.T_CtrleAction.udiErrorID:=0;
			xMoveContinousVel:=FALSE;
		(* axis not ready *)
		95:	T_Visu.ptrT_ExchgParam^.T_StationCommon.wState:=T_Visu.ptrT_ExchgParam^.T_StationCommon.wState AND 16#BF;
			TimerNotReady(IN:=TRUE);
			xMoveContinousVel:=FALSE;
		(* error *)
		99:	T_Visu.ptrT_ExchgParam^.T_StationCommon.wState:=T_Visu.ptrT_ExchgParam^.T_StationCommon.wState AND 16#BF;
			T_Visu.T_CtrleAction.xDone:=TRUE;
			T_Visu.T_CtrleAction.xNotReady:=FALSE;
			IF (ptrTeachINAxis^.T_Config_Gen.iTyp <> 0) THEN
				diErrorNr:=(ptrTeachINAxis^.T_Config_Gen.iTyp * 1000000) + ptrTeachINAxis^.T_CtrleSingle.udiErrorID;
			ELSE
				diErrorNr:=0;
			END_IF;
			FBErrorMessage(	diErrorNr:=diErrorNr,
							T_ErrorList:=T_ErrorList);
			T_Visu.ptrT_ExchgParam^.T_Visu.T_Message.sDynamicTextEnglish:=FBErrorMessage.sErrorTextEnglish;
			T_Visu.ptrT_ExchgParam^.T_Visu.T_Message.sDynamicTextDeutsch:=FBErrorMessage.sErrorTextDeutsch;
			T_Visu.ptrT_ExchgParam^.T_Visu.T_Message.sDynamicTextFrancais:=FBErrorMessage.sErrorTextFrancais;
			T_Visu.ptrT_ExchgParam^.T_SafetyCtrl.xSetForceError:=TRUE;
			T_Visu.ptrT_ExchgParam^.T_SafetyCtrl.diSetForceErrorNr:=diErrorNr;
			T_Visu.T_CtrleAction.xErr:=FALSE;
			T_Visu.T_CtrleAction.udiErrorID:=0;
			ptrTeachINAxis^.T_CtrleSingle.iFunction:=1;
			ptrTeachINAxis^.T_CtrleSingle.xExecute:=TRUE;
			xMoveContinousVel:=FALSE;
		END_CASE
	END_IF

(* Action Toggle Axis Power *)
	IF xToggleAxisPower OR xResetAxis THEN
		(* Step toggle Axis power *)
		CASE iStepAction OF
		(* check axis *)
		1:	IF NOT T_Station.TControl.xHardwareConfigError THEN
				xStepActionDone:=FALSE;
				iStepAction:=95;
				IF xToggleAxisPower THEN
					xTmp:=	ptrTeachINAxis^.T_CtrleSingle.xDone
							AND ptrTeachINAxis^.T_CtrleSingle.xNotMoving
							AND NOT(ptrTeachINAxis^.T_CtrleSingle.xErr)
							AND NOT(ptrTeachINAxis^.T_CtrleSingle.xExecute);
				END_IF;
				IF xResetAxis THEN
					xTmp:=	(ptrTeachINAxis^.T_CtrleSingle.xDone OR ptrTeachINAxis^.T_CtrleSingle.xErr)
							AND ptrTeachINAxis^.T_CtrleSingle.xNotMoving
							AND NOT(ptrTeachINAxis^.T_CtrleSingle.xExecute);
				END_IF;
				(* Start/Stop position or speed of teachin page has to be confirmed *)
				IF xTmp THEN
					iStepAction:=10;
				END_IF
			ELSE
				iStepAction:=95;
			END_IF;
		(* activ function axis *)
		10:	bStateMachine:=2;
			xSetStateMachine:=TRUE;
			IF xToggleAxisPower THEN
				IF ptrTeachINAxis^.T_CtrleSingle.xPower THEN
					ptrTeachINAxis^.T_CtrleSingle.iFunction:=4;
				END_IF;
				IF NOT(ptrTeachINAxis^.T_CtrleSingle.xPower) THEN
					ptrTeachINAxis^.T_CtrleSingle.iFunction:=3;
				END_IF;
			END_IF;
			IF xResetAxis THEN
				ptrTeachINAxis^.T_CtrleSingle.iFunction:=1;
			END_IF;
			ptrTeachINAxis^.T_CtrleSingle.xExecute:=TRUE;
			(* next step *)
			iStepAction:=20;
			xStepActionDone:=FALSE;
		(* confirm execution *)
		20:	IF NOT(xStepActionDone) THEN
			(* confirm execution *)
				ptrTeachINAxis^.T_CtrleSingle.xExecute:=FALSE;
				xStepActionDone:=TRUE;
			ELSE
				IF ptrTeachINAxis^.T_CtrleSingle.xDone THEN
				(* confirm action next step *)
					bStateMachine:=1;
					xSetStateMachine:=TRUE;
					iStepAction:=90;
					xStepActionDone:=FALSE;
				ELSE
					IF ptrTeachINAxis^.T_CtrleSingle.xErr THEN
					(* activ action not ready or error *)
						iStepAction:=99;
						xStepActionDone:=FALSE;
					END_IF
				END_IF
			END_IF
		(* action done *)
		90:	T_Visu.ptrT_ExchgParam^.T_StationCommon.wState:=T_Visu.ptrT_ExchgParam^.T_StationCommon.wState AND 16#BF;
			T_Visu.T_CtrleAction.xDone:=TRUE;
			T_Visu.T_CtrleAction.xNotReady:=FALSE;
			T_Visu.T_CtrleAction.xErr:=FALSE;
			T_Visu.T_CtrleAction.udiErrorID:=0;
			xToggleAxisPower:=xResetAxis:=FALSE;
		(* axis not ready *)
		95:	T_Visu.ptrT_ExchgParam^.T_StationCommon.wState:=T_Visu.ptrT_ExchgParam^.T_StationCommon.wState AND 16#BF;
			TimerNotReady(IN:=TRUE);
			xToggleAxisPower:=xResetAxis:=FALSE;
		(* error *)
		99:	T_Visu.ptrT_ExchgParam^.T_StationCommon.wState:=T_Visu.ptrT_ExchgParam^.T_StationCommon.wState AND 16#BF;
			T_Visu.T_CtrleAction.xDone:=TRUE;
			T_Visu.T_CtrleAction.xNotReady:=FALSE;
			IF (ptrTeachINAxis^.T_Config_Gen.iTyp <> 0) THEN
				diErrorNr:=(ptrTeachINAxis^.T_Config_Gen.iTyp * 1000000) + ptrTeachINAxis^.T_CtrleSingle.udiErrorID;
			ELSE
				diErrorNr:=0;
			END_IF;
			FBErrorMessage(	diErrorNr:=diErrorNr,
							T_ErrorList:=T_ErrorList);
			T_Visu.ptrT_ExchgParam^.T_Visu.T_Message.sDynamicTextEnglish:=FBErrorMessage.sErrorTextEnglish;
			T_Visu.ptrT_ExchgParam^.T_Visu.T_Message.sDynamicTextDeutsch:=FBErrorMessage.sErrorTextDeutsch;
			T_Visu.ptrT_ExchgParam^.T_Visu.T_Message.sDynamicTextFrancais:=FBErrorMessage.sErrorTextFrancais;
			T_Visu.ptrT_ExchgParam^.T_SafetyCtrl.xSetForceError:=TRUE;
			T_Visu.ptrT_ExchgParam^.T_SafetyCtrl.diSetForceErrorNr:=diErrorNr;
			T_Visu.T_CtrleAction.xErr:=FALSE;
			T_Visu.T_CtrleAction.udiErrorID:=0;
			ptrTeachINAxis^.T_CtrleSingle.iFunction:=1;
			ptrTeachINAxis^.T_CtrleSingle.xExecute:=TRUE;
			xToggleAxisPower:=xResetAxis:=FALSE;
		END_CASE
	END_IF

(* Reference axis *)
	IF xReferenceAxis THEN
		(* Step reference Axis *)
		CASE iStepAction OF
		(* check axis *)
		1:	IF NOT T_Station.TControl.xHardwareConfigError THEN
				xStepActionDone:=FALSE;
				iStepAction:=95;
				xTmp:=	T_Station.THardware.TAxisToolFeeder.T_CtrleSingle.xDone
						AND T_Station.THardware.TAxisToolFeeder.T_CtrleSingle.xPower
						AND T_Station.THardware.TAxisToolFeeder.T_CtrleSingle.xNotMoving
						AND NOT(T_Station.THardware.TAxisToolFeeder.T_CtrleSingle.xErr)
						AND NOT(T_Station.THardware.TAxisToolFeeder.T_CtrleSingle.xExecute);
				(* Start/Stop position or speed of teachin page has to be confirmed *)
				IF xTmp THEN
					iStepAction:=10;
				END_IF
			ELSE
				iStepAction:=95;
			END_IF;
		(* activ function axis *)
		10:	bStateMachine:=2;
			xSetStateMachine:=TRUE;
			T_Station.THardware.TAxisToolFeeder.T_CtrleSingle.lrHomingMethode:=5;
			T_Station.THardware.TAxisToolFeeder.T_CtrleSingle.lrHomeOffset:=0.0;
			T_Station.THardware.TAxisToolFeeder.T_CtrleSingle.lrHomeSpeedSwitch:=T_NovRAM.T_Data.T_Standard.T_TeachINToolFeeder.rRefSpeed;
			T_Station.THardware.TAxisToolFeeder.T_CtrleSingle.lrHomeSpeedZero:=T_NovRAM.T_Data.T_Standard.T_TeachINToolFeeder.rRefSpeed / 10.0;
			T_Station.THardware.TAxisToolFeeder.T_CtrleSingle.lrHomeAcceleration:=T_NovRAM.T_Data.T_Standard.T_TeachINToolFeeder.rAcceleration;
			T_Station.THardware.TAxisToolFeeder.T_CtrleSingle.iFunction:=9;	(* Reference Axis *)
			T_Station.THardware.TAxisToolFeeder.T_CtrleSingle.xExecute:=TRUE;
			(* next step *)
			iStepAction:=20;
			xStepActionDone:=FALSE;
		(* confirm execution *)
		20:	IF NOT(xStepActionDone) THEN
			(* confirm execution *)
				T_Station.THardware.TAxisToolFeeder.T_CtrleSingle.xExecute:=FALSE;
				xStepActionDone:=TRUE;
			ELSE
				IF T_Station.THardware.TAxisToolFeeder.T_CtrleSingle.xDone THEN
				(* confirm action next step *)
					bStateMachine:=1;
					xSetStateMachine:=TRUE;
					iStepAction:=90;
					xStepActionDone:=FALSE;
				ELSE
					IF T_Station.THardware.TAxisToolFeeder.T_CtrleSingle.xErr THEN
					(* activ action not ready or error *)
						iStepAction:=99;
						xStepActionDone:=FALSE;
					END_IF
				END_IF
			END_IF
		(* action done *)
		90:	T_Visu.ptrT_ExchgParam^.T_StationCommon.wState:=T_Visu.ptrT_ExchgParam^.T_StationCommon.wState AND 16#BF;
			T_Visu.T_CtrleAction.xDone:=TRUE;
			T_Visu.T_CtrleAction.xNotReady:=FALSE;
			T_Visu.T_CtrleAction.xErr:=FALSE;
			T_Visu.T_CtrleAction.udiErrorID:=0;
			xReferenceAxis:=FALSE;
		(* axis not ready *)
		95:	T_Visu.ptrT_ExchgParam^.T_StationCommon.wState:=T_Visu.ptrT_ExchgParam^.T_StationCommon.wState AND 16#BF;
			TimerNotReady(IN:=TRUE);
			xReferenceAxis:=FALSE;
		(* error *)
		99:	T_Visu.ptrT_ExchgParam^.T_StationCommon.wState:=T_Visu.ptrT_ExchgParam^.T_StationCommon.wState AND 16#BF;
			T_Visu.T_CtrleAction.xDone:=TRUE;
			T_Visu.T_CtrleAction.xNotReady:=FALSE;
			IF (T_Station.THardware.TAxisToolFeeder.T_Config_Gen.iTyp <> 0) THEN
				diErrorNr:=(T_Station.THardware.TAxisToolFeeder.T_Config_Gen.iTyp * 1000000) + T_Station.THardware.TAxisToolFeeder.T_CtrleSingle.udiErrorID;
			ELSE
				diErrorNr:=0;
			END_IF;
			FBErrorMessage(	diErrorNr:=diErrorNr,
							T_ErrorList:=T_ErrorList);
			T_Visu.ptrT_ExchgParam^.T_Visu.T_Message.sDynamicTextEnglish:=FBErrorMessage.sErrorTextEnglish;
			T_Visu.ptrT_ExchgParam^.T_Visu.T_Message.sDynamicTextDeutsch:=FBErrorMessage.sErrorTextDeutsch;
			T_Visu.ptrT_ExchgParam^.T_Visu.T_Message.sDynamicTextFrancais:=FBErrorMessage.sErrorTextFrancais;
			T_Visu.ptrT_ExchgParam^.T_SafetyCtrl.xSetForceError:=TRUE;
			T_Visu.ptrT_ExchgParam^.T_SafetyCtrl.diSetForceErrorNr:=diErrorNr;
			T_Visu.T_CtrleAction.xErr:=FALSE;
			T_Visu.T_CtrleAction.udiErrorID:=0;
			T_Station.THardware.TAxisToolFeeder.T_CtrleSingle.iFunction:=1;
			T_Station.THardware.TAxisToolFeeder.T_CtrleSingle.xExecute:=TRUE;
			xReferenceAxis:=FALSE;
		END_CASE
	END_IF

(* Teach axis Position *)
	IF xTeachPosition THEN
		CASE iStepAction OF
		(* check axis *)
		1:	IF NOT T_Station.TControl.xHardwareConfigError THEN
				xStepActionDone:=FALSE;
				iStepAction:=10;
			ELSE
				iStepAction:=95;
			END_IF;
		(* Check teachin position *)
		10:	IF (iSelectedAxis = 4) THEN
				IF (T_Visu.ptrT_ExchgParam^.T_TeachIn.iSaveToolFeederPos = 0) THEN
				(* Display message 'Move position can not be teached' *)
					tTimeOutAction:=TimerAction.ET+T#2s;
					T_Visu.ptrT_ExchgParam^.T_Visu.T_Message.iState:=31;
					(* Action has been cancelled *)
					iStepAction:=89;
				ELSE
					iStepAction:=20;
				END_IF
			END_IF;
			IF (iSelectedAxis = 5) THEN
				IF (T_Visu.ptrT_ExchgParam^.T_TeachIn.iSaveGrindFeederPos = 0) THEN
				(* Display message 'Move position can not be teached' *)
					tTimeOutAction:=TimerAction.ET+T#2s;
					T_Visu.ptrT_ExchgParam^.T_Visu.T_Message.iState:=31;
					(* Action has been cancelled *)
					iStepAction:=89;
				(* Software limit switch pos and neg not possible that we can teach this position *)
				ELSIF (T_Visu.ptrT_ExchgParam^.T_TeachIn.iSaveGrindFeederPos = 3) OR (T_Visu.ptrT_ExchgParam^.T_TeachIn.iSaveGrindFeederPos = 4) THEN
				(* Display message 'Selected position can not be teached' *)
					tTimeOutAction:=TimerAction.ET+T#2s;
					T_ExchgParam.T_Visu.T_Message.iState:=30;
					(* Action has been cancelled *)
					iStepAction:=89;
				ELSE
					iStepAction:=20;
				END_IF
			END_IF;
		(* Check if the Axis is referenced *)
		20:	IF (iSelectedAxis = 4) THEN
				xTmp:=	T_Station.TControl.xReferenced;
				IF NOT(xTmp) THEN
					(* Display message 'Axis not referenced' *)
					tTimeOutAction:=TimerAction.ET+T#2s;
					T_Visu.ptrT_ExchgParam^.T_Visu.T_Message.iState:=18;
					(* Action has been cancelled *)
					iStepAction:=89;
				ELSE
					iStepAction:=30;
				END_IF;
			ELSE
				iStepAction:=30;
			END_IF;
		(* Display message to ask for confirmation *)
		30:	T_Visu.ptrT_ExchgParam^.T_Visu.T_Message.iState:=108;
			iStepAction:=40;
		(* waiting for key <Enter> or <Esc> *)
		40:	IF RisingEdgeKeyPanel_Enter.Q THEN iStepAction:=50;
			ELSE IF RisingEdgeKeyPanel_Esc.Q THEN iStepAction:=90; END_IF END_IF
			(* An other message has been displayed, stop teach action *)
			IF T_Visu.ptrT_ExchgParam^.T_Visu.T_Message.iState<>108 THEN iStepAction:=90; END_IF
		50:	IF (iSelectedAxis = 4) AND (T_Visu.ptrT_ExchgParam^.T_TeachIn.iSaveToolFeederPos = 1) THEN
				T_Visu.ptrT_ExchgParam^.T_StationCommon.T_ProcessPara.rStartPosToolFeedAuto:=
					LREAL_TO_REAL(ptrTeachINAxis^.T_LiveValue.lrActualPosition);
			ELSIF (iSelectedAxis = 4) AND (T_Visu.ptrT_ExchgParam^.T_TeachIn.iSaveToolFeederPos = 2) THEN
				T_Visu.ptrT_ExchgParam^.T_StationCommon.T_CalibrationPara.rStartPosToolFeedCalib:=
					LREAL_TO_REAL(ptrTeachINAxis^.T_LiveValue.lrActualPosition);
			ELSIF (iSelectedAxis = 4) AND (T_Visu.ptrT_ExchgParam^.T_TeachIn.iSaveToolFeederPos = 3) THEN
				T_Visu.ptrT_ExchgParam^.T_StationCommon.T_CalibrationPara.rMeasurePosToolFeedCalib:=
					LREAL_TO_REAL(ptrTeachINAxis^.T_LiveValue.lrActualPosition);
			ELSIF (iSelectedAxis = 4) AND (T_Visu.ptrT_ExchgParam^.T_TeachIn.iSaveToolFeederPos = 4) THEN
				T_Visu.ptrT_ExchgParam^.T_TeachIn.TParam_AxisPosition.rLoadPosToolFeedAuto:=
					LREAL_TO_REAL(ptrTeachINAxis^.T_LiveValue.lrActualPosition);
			END_IF;
			iStepAction:=60;
			IF (iSelectedAxis = 5) AND (T_Visu.ptrT_ExchgParam^.T_TeachIn.iSaveGrindFeederPos = 1) THEN
				(* The StartPosition will be set as absolut position for the GrindFeeder Axis *)
				T_Station.THardware.TAxisGrindFeeder.T_CtrleSingle.rSetPosition:=
					T_NovRam.T_Data.T_ProcessImageData.T_ProcessPara.rToolDiameterProcess;
				iStepAction:=80;
			END_IF;
			IF (iSelectedAxis = 5) AND (T_Visu.ptrT_ExchgParam^.T_TeachIn.iSaveGrindFeederPos = 2) THEN
				(* The Security Position will be set as absolut position for the GrindFeeder Axis *)
				T_Station.THardware.TAxisGrindFeeder.T_CtrleSingle.rSetPosition:=
										T_NovRam.T_Data.T_ProcessImageData.T_ProcessPara.rToolDiameterProcess +
										T_NovRam.T_Data.T_ProcessImageData.T_ProcessPara.rSecurityPosGrindFeedProcess;
				iStepAction:=80;
			END_IF;
		60:	xAction_SaveNovRAMWithoutConfirm:=TRUE;
			iStepActionNovRam:=1;
			(* next step *)
			iStepAction:=70;
		70:	IF NOT(xAction_SaveNovRAMWithoutConfirm) THEN
				iStepAction:=90;
			END_IF;
		(* activ function axis *)
		80:	T_Station.THardware.TAxisGrindFeeder.T_CtrleSingle.iFunction:=11;
			T_Station.THardware.TAxisGrindFeeder.T_CtrleSingle.xExecute:=TRUE;
			(* next step *)
			iStepAction:=81;
			xStepActionDone:=FALSE;
		(* confirm execution *)
		81:	IF NOT(xStepActionDone) THEN
			(* confirm execution *)
				T_Station.THardware.TAxisGrindFeeder.T_CtrleSingle.xExecute:=FALSE;
				xStepActionDone:=TRUE;
			ELSE
				IF T_Station.THardware.TAxisGrindFeeder.T_CtrleSingle.xDone THEN
				(* confirm action next step *)
					iStepAction:=90;
					xStepActionDone:=FALSE;
				ELSE
					IF T_Station.THardware.TAxisGrindFeeder.T_CtrleSingle.xErr THEN
					(* activ action not ready or error *)
						iStepAction:=98;
						xStepActionDone:=FALSE;
					END_IF
				END_IF
			END_IF
		(* waiting timeout *)
		89: IF TimerAction.Q THEN iStepAction:=90; END_IF
		(* axis not ready *)
		95:	TimerNotReady(IN:=TRUE);
			xTeachPosition:=FALSE;
		(* slow/fast configuration done *)
		90:	T_Visu.T_CtrleAction.xDone:=TRUE;
			T_Visu.T_CtrleAction.xNotReady:=FALSE;
			T_Visu.T_CtrleAction.xErr:=FALSE;
			T_Visu.T_CtrleAction.udiErrorID:=0;
			xTeachPosition:=FALSE;
		(* axis error *)
		98:	T_Visu.ptrT_ExchgParam^.T_StationCommon.wState:=T_Visu.ptrT_ExchgParam^.T_StationCommon.wState AND 16#BF;
			T_Visu.T_CtrleAction.xDone:=TRUE;
			T_Visu.T_CtrleAction.xNotReady:=FALSE;
			IF (T_Station.THardware.TAxisGrindFeeder.T_Config_Gen.iTyp <> 0) THEN
				diErrorNr:=(T_Station.THardware.TAxisGrindFeeder.T_Config_Gen.iTyp * 1000000) + T_Station.THardware.TAxisGrindFeeder.T_CtrleSingle.udiErrorID;
			ELSE
				diErrorNr:=0;
			END_IF;
			FBErrorMessage(	diErrorNr:=diErrorNr,
							T_ErrorList:=T_ErrorList);
			T_Visu.ptrT_ExchgParam^.T_Visu.T_Message.sDynamicTextEnglish:=FBErrorMessage.sErrorTextEnglish;
			T_Visu.ptrT_ExchgParam^.T_Visu.T_Message.sDynamicTextDeutsch:=FBErrorMessage.sErrorTextDeutsch;
			T_Visu.ptrT_ExchgParam^.T_Visu.T_Message.sDynamicTextFrancais:=FBErrorMessage.sErrorTextFrancais;
			T_Visu.ptrT_ExchgParam^.T_SafetyCtrl.xSetForceError:=TRUE;
			T_Visu.ptrT_ExchgParam^.T_SafetyCtrl.diSetForceErrorNr:=diErrorNr;
			T_Visu.T_CtrleAction.xErr:=FALSE;
			T_Visu.T_CtrleAction.udiErrorID:=0;
			T_Station.THardware.TAxisGrindFeeder.T_CtrleSingle.iFunction:=1;
			T_Station.THardware.TAxisGrindFeeder.T_CtrleSingle.xExecute:=TRUE;
			xTeachPosition:=FALSE;
		99:	T_Visu.T_CtrleAction.xDone:=FALSE;
			T_Visu.T_CtrleAction.xNotReady:=FALSE;
			T_Visu.T_CtrleAction.xErr:=TRUE;
			T_Visu.T_CtrleAction.udiErrorID:=16#F0000 + T_Visu.T_CtrleAction.iFunction;
			xTeachPosition:=FALSE;
		END_CASE
	END_IF

(* Calculate the position between the RefIndex and the RefSensor *)
	IF xCalcAngleRefIndex THEN
		(* Step calc the position between the RefIndex and the RefSensor *)
		CASE iStepAction OF
		(* check axis *)
		1:	IF NOT T_Station.TControl.xHardwareConfigError THEN
				xStepActionDone:=FALSE;
				iStepAction:=10;
			ELSE
				iStepAction:=95;
			END_IF;
		(* check axis state *)
		10:	xStepActionDone:=FALSE;
			xTmp:=	T_Station.THardware.TAxisToolFeeder.T_CtrleSingle.xDone
					AND T_Station.THardware.TAxisToolFeeder.T_CtrleSingle.xReady
					AND T_Station.THardware.TAxisToolFeeder.T_CtrleSingle.xNotMoving
					AND NOT(T_Station.THardware.TAxisToolFeeder.T_CtrleSingle.xErr)
					AND NOT(T_Station.THardware.TAxisToolFeeder.T_CtrleSingle.xExecute);
			IF xTmp THEN
				iStepAction:=20;
			ELSE
				iStepAction:=95;
			END_IF
		(* activ function axis *)
		20:	bStateMachine:=2;
			xSetStateMachine:=TRUE;
			T_Station.THardware.TAxisToolFeeder.T_CtrleSingle.lrHomingMethode:=5;
			T_Station.THardware.TAxisToolFeeder.T_CtrleSingle.lrHomeOffset:=0.0;
			T_Station.THardware.TAxisToolFeeder.T_CtrleSingle.lrHomeSpeedSwitch:=T_NovRAM.T_Data.T_Standard.T_TeachINToolFeeder.rRefSpeed;
			T_Station.THardware.TAxisToolFeeder.T_CtrleSingle.lrHomeSpeedZero:=T_NovRAM.T_Data.T_Standard.T_TeachINToolFeeder.rRefSpeed / 10.0;
			T_Station.THardware.TAxisToolFeeder.T_CtrleSingle.lrHomeAcceleration:=T_NovRAM.T_Data.T_Standard.T_TeachINToolFeeder.rAcceleration;
			T_Station.THardware.TAxisToolFeeder.T_CtrleSingle.lrDecceleration:=T_NovRAM.T_Data.T_Standard.T_TeachINToolFeeder.rDeceleration;
			T_Station.THardware.TAxisToolFeeder.T_CtrleSingle.lrVelocity:=0.1;
			T_Station.THardware.TAxisToolFeeder.T_CtrleSingle.lrPosition:=0;
			T_Station.THardware.TAxisToolFeeder.T_CtrleSingle.lrDistance:=-2;
			T_Station.THardware.TAxisToolFeeder.T_CtrleSingle.iFunction:=19;
			T_Station.THardware.TAxisToolFeeder.T_CtrleSingle.xExecute:=TRUE;
			(* next step *)
			iStepAction:=30;
			xStepActionDone:=FALSE;
		(* confirm execution *)
		30:	IF NOT(xStepActionDone) THEN
			(* confirm execution *)
				T_Station.THardware.TAxisToolFeeder.T_CtrleSingle.xExecute:=FALSE;
				xStepActionDone:=TRUE;
			ELSE
				IF T_Station.THardware.TAxisToolFeeder.T_CtrleSingle.xDone THEN
					T_Visu.ptrT_ExchgParam^.T_StationCommon.iWireFeederAngleRefIndex:=T_Station.THardware.TAxisToolFeeder.T_CtrleSingle.iStrokeAngleRefIndex;
					xStepActionDone:=FALSE;
					iStepAction:=40;
				ELSE
					IF T_Station.THardware.TAxisToolFeeder.T_CtrleSingle.xErr THEN
					(* activ action not ready or error *)
						iStepAction:=99;
						xStepActionDone:=FALSE;
					END_IF
				END_IF
			END_IF;
		(* Reference axis *)
		40:	T_Station.THardware.TAxisToolFeeder.T_CtrleSingle.lrHomingMethode:=5;
			T_Station.THardware.TAxisToolFeeder.T_CtrleSingle.lrHomeOffset:=0.0;
			T_Station.THardware.TAxisToolFeeder.T_CtrleSingle.lrHomeSpeedSwitch:=T_NovRAM.T_Data.T_Standard.T_TeachINToolFeeder.rRefSpeed;
			T_Station.THardware.TAxisToolFeeder.T_CtrleSingle.lrHomeSpeedZero:=T_NovRAM.T_Data.T_Standard.T_TeachINToolFeeder.rRefSpeed / 10.0;
			T_Station.THardware.TAxisToolFeeder.T_CtrleSingle.lrHomeAcceleration:=T_NovRAM.T_Data.T_Standard.T_TeachINToolFeeder.rAcceleration;
			T_Station.THardware.TAxisToolFeeder.T_CtrleSingle.iFunction:=9;	(* Reference Axis *)
			T_Station.THardware.TAxisToolFeeder.T_CtrleSingle.xExecute:=TRUE;
			(* next step *)
			iStepAction:=50;
			xStepActionDone:=FALSE;
		(* confirm execution *)
		50:	IF NOT(xStepActionDone) THEN
			(* confirm execution *)
				T_Station.THardware.TAxisToolFeeder.T_CtrleSingle.xExecute:=FALSE;
				xStepActionDone:=TRUE;
			ELSE
				IF T_Station.THardware.TAxisToolFeeder.T_CtrleSingle.xDone THEN
				(* confirm action next step *)
					bStateMachine:=1;
					xSetStateMachine:=TRUE;
					iStepAction:=90;
					xStepActionDone:=FALSE;
				ELSE
					IF T_Station.THardware.TAxisToolFeeder.T_CtrleSingle.xErr THEN
					(* activ action not ready or error *)
						iStepAction:=99;
						xStepActionDone:=FALSE;
					END_IF
				END_IF
			END_IF
		(* waiting time out *)
		89:	IF TimerAction.Q THEN iStepAction:=90; END_IF
		(* action done *)
		90:	T_Visu.T_CtrleAction.xDone:=TRUE;
			T_Visu.T_CtrleAction.xNotReady:=FALSE;
			T_Visu.T_CtrleAction.xErr:=FALSE;
			T_Visu.T_CtrleAction.udiErrorID:=0;
			xCalcAngleRefIndex:=FALSE;
		(* axis not ready *)
		95:	TimerNotReady(IN:=TRUE);
			xCalcAngleRefIndex:=FALSE;
		(* error *)
		99:	T_Visu.ptrT_ExchgParam^.T_StationCommon.wState:=T_Visu.ptrT_ExchgParam^.T_StationCommon.wState AND 16#BF;
			T_Visu.T_CtrleAction.xDone:=TRUE;
			T_Visu.T_CtrleAction.xNotReady:=FALSE;
			IF (T_Station.THardware.TAxisToolFeeder.T_Config_Gen.iTyp <> 0) THEN
				diErrorNr:=(T_Station.THardware.TAxisToolFeeder.T_Config_Gen.iTyp * 1000000) + T_Station.THardware.TAxisToolFeeder.T_CtrleSingle.udiErrorID;
			ELSE
				diErrorNr:=0;
			END_IF;
			FBErrorMessage(	diErrorNr:=diErrorNr,
							T_ErrorList:=T_ErrorList);
			T_Visu.ptrT_ExchgParam^.T_Visu.T_Message.sDynamicTextEnglish:=FBErrorMessage.sErrorTextEnglish;
			T_Visu.ptrT_ExchgParam^.T_Visu.T_Message.sDynamicTextDeutsch:=FBErrorMessage.sErrorTextDeutsch;
			T_Visu.ptrT_ExchgParam^.T_Visu.T_Message.sDynamicTextFrancais:=FBErrorMessage.sErrorTextFrancais;
			T_Visu.ptrT_ExchgParam^.T_SafetyCtrl.xSetForceError:=TRUE;
			T_Visu.ptrT_ExchgParam^.T_SafetyCtrl.diSetForceErrorNr:=diErrorNr;
			T_Visu.T_CtrleAction.xErr:=FALSE;
			T_Visu.T_CtrleAction.udiErrorID:=0;
			T_Station.THardware.TAxisToolFeeder.T_CtrleSingle.iFunction:=1;
			T_Station.THardware.TAxisToolFeeder.T_CtrleSingle.xExecute:=TRUE;
			xCalcAngleRefIndex:=FALSE;
		END_CASE
	END_IF;

(* Switch ToolRotation Master Slave *)
	IF xSwitchMasterSlave THEN
		CASE iStepAction OF
		(* check axis *)
		1:	IF NOT T_Station.TControl.xHardwareConfigError THEN
				xStepActionDone:=FALSE;
				iStepAction:=95;
				xTmp:=	T_Station.THardware.TAxisToolLeft.T_CtrleSingle.xDone AND
						T_Station.THardware.TAxisToolLeft.T_CtrleSingle.xNotMoving AND
						NOT(T_Station.THardware.TAxisToolLeft.T_CtrleSingle.xErr) AND
						NOT(T_Station.THardware.TAxisToolLeft.T_CtrleSingle.xExecute);
				xTmp:=	xTmp AND
						((T_Station.THardware.TAxisToolCenter.T_CtrleSingle.xDone AND
						T_Station.THardware.TAxisToolCenter.T_CtrleSingle.xNotMoving AND
						NOT(T_Station.THardware.TAxisToolCenter.T_CtrleSingle.xErr) AND
						NOT(T_Station.THardware.TAxisToolCenter.T_CtrleSingle.xExecute) AND
						xMicroRodActive) OR
						NOT(xMicroRodActive));
				xTmp:=	xTmp AND
						T_Station.THardware.TAxisToolRight.T_CtrleSingle.xDone AND
						T_Station.THardware.TAxisToolRight.T_CtrleSingle.xNotMoving AND
						NOT(T_Station.THardware.TAxisToolRight.T_CtrleSingle.xErr) AND
						NOT(T_Station.THardware.TAxisToolRight.T_CtrleSingle.xExecute);
				xTmp:=	xTmp AND
						((T_Station.THardware.TAxisToolFeeder.T_CtrleSingle.xDone AND
						T_Station.THardware.TAxisToolFeeder.T_CtrleSingle.xNotMoving AND
						NOT(T_Station.THardware.TAxisToolFeeder.T_CtrleSingle.xErr) AND
						NOT(T_Station.THardware.TAxisToolFeeder.T_CtrleSingle.xExecute) AND
						NOT(xMicroRodActive)) OR
						xMicroRodActive);
				(* Start/Stop position or speed of teachin page has to be confirmed *)
				IF xTmp THEN
					iStepAction:=10;
				END_IF
			ELSE
				iStepAction:=95;
			END_IF;
		(* activ function axis *)
		10:	bStateMachine:=2;
			xSetStateMachine:=TRUE;
			T_Station.THardware.TAxisToolRight.T_CtrleSingle.iFunction:=25;
			T_Station.THardware.TAxisToolRight.T_CtrleSingle.xExecute:=TRUE;
			IF xMicroRodActive THEN
				T_Station.THardware.TAxisToolCenter.T_CtrleSingle.iFunction:=25;
				T_Station.THardware.TAxisToolCenter.T_CtrleSingle.xExecute:=TRUE;
			END_IF;
			IF NOT(xMicroRodActive) THEN
				T_Station.THardware.TAxisToolFeeder.T_CtrleSingle.iFunction:=25;
				T_Station.THardware.TAxisToolFeeder.T_CtrleSingle.xExecute:=TRUE;
			END_IF;
			(* next step *)
			iStepAction:=20;
			xStepActionDone:=FALSE;
		(* confirm execution *)
		20:	IF NOT(xStepActionDone) THEN
			(* confirm execution *)
				T_Station.THardware.TAxisToolRight.T_CtrleSingle.xExecute:=FALSE;
				IF xMicroRodActive THEN
					T_Station.THardware.TAxisToolCenter.T_CtrleSingle.xExecute:=FALSE;
				END_IF;
				IF NOT(xMicroRodActive) THEN
					T_Station.THardware.TAxisToolFeeder.T_CtrleSingle.xExecute:=FALSE;
				END_IF;
				xStepActionDone:=TRUE;
			ELSE
				IF T_Station.THardware.TAxisToolRight.T_CtrleSingle.xDone AND ((T_Station.THardware.TAxisToolCenter.T_CtrleSingle.xDone AND xMicroRodActive) OR NOT(xMicroRodActive)) AND
				     ((T_Station.THardware.TAxisToolFeeder.T_CtrleSingle.xDone AND NOT(xMicroRodActive)) OR xMicroRodActive) THEN
				(* confirm action next step *)
					IF T_Station.THardware.TAxisToolRight.T_CtrleSingle.xSlave AND T_Station.THardware.TAxisToolCenter.T_CtrleSingle.xSlave AND xMicroRodActive THEN
						xToolRotationMasterSlave:=TRUE;
					END_IF;
					IF NOT(T_Station.THardware.TAxisToolRight.T_CtrleSingle.xSlave) AND NOT(T_Station.THardware.TAxisToolCenter.T_CtrleSingle.xSlave) AND xMicroRodActive THEN
						xToolRotationMasterSlave:=FALSE;
					END_IF;
					IF T_Station.THardware.TAxisToolRight.T_CtrleSingle.xSlave AND T_Station.THardware.TAxisToolFeeder.T_CtrleSingle.xSlave AND NOT(xMicroRodActive) THEN
						xToolRotationMasterSlave:=TRUE;
					END_IF;
					IF NOT(T_Station.THardware.TAxisToolRight.T_CtrleSingle.xSlave) AND NOT(T_Station.THardware.TAxisToolFeeder.T_CtrleSingle.xSlave) AND NOT(xMicroRodActive) THEN
						xToolRotationMasterSlave:=FALSE;
					END_IF;
					iStepAction:=90;
					xStepActionDone:=FALSE;
				ELSE
					IF T_Station.THardware.TAxisToolRight.T_CtrleSingle.xErr OR (T_Station.THardware.TAxisToolCenter.T_CtrleSingle.xErr AND xMicroRodActive) OR
					     (T_Station.THardware.TAxisToolFeeder.T_CtrleSingle.xErr AND NOT(xMicroRodActive)) THEN
					(* activ action not ready or error *)
						iStepAction:=99;
						xStepActionDone:=FALSE;
					END_IF
				END_IF
			END_IF
		(* action done *)
		90:	bStateMachine:=1;
			xSetStateMachine:=TRUE;
			T_Visu.ptrT_ExchgParam^.T_StationCommon.wState:=T_Visu.ptrT_ExchgParam^.T_StationCommon.wState AND 16#BF;
			T_Visu.T_CtrleAction.xDone:=TRUE;
			T_Visu.T_CtrleAction.xNotReady:=FALSE;
			T_Visu.T_CtrleAction.xErr:=FALSE;
			T_Visu.T_CtrleAction.udiErrorID:=0;
			xSwitchMasterSlave:=FALSE;
		(* axis not ready *)
		95:	T_Visu.ptrT_ExchgParam^.T_StationCommon.wState:=T_Visu.ptrT_ExchgParam^.T_StationCommon.wState AND 16#BF;
			TimerNotReady(IN:=TRUE);
			xSwitchMasterSlave:=FALSE;
		(* error *)
		99:	T_Visu.ptrT_ExchgParam^.T_StationCommon.wState:=T_Visu.ptrT_ExchgParam^.T_StationCommon.wState AND 16#BF;
			T_Visu.T_CtrleAction.xDone:=TRUE;
			T_Visu.T_CtrleAction.xNotReady:=FALSE;
			IF T_Station.THardware.TAxisToolRight.T_CtrleSingle.xErr THEN
				IF (T_Station.THardware.TAxisToolRight.T_Config_Gen.iTyp <> 0) THEN
					diErrorNr:=(T_Station.THardware.TAxisToolRight.T_Config_Gen.iTyp * 1000000) + T_Station.THardware.TAxisToolRight.T_CtrleSingle.udiErrorID;
				ELSE
					diErrorNr:=0;
				END_IF;
			END_IF;
			IF T_Station.THardware.TAxisToolCenter.T_CtrleSingle.xErr AND xMicroRodActive THEN
				IF (T_Station.THardware.TAxisToolCenter.T_Config_Gen.iTyp <> 0) THEN
					diErrorNr:=(T_Station.THardware.TAxisToolCenter.T_Config_Gen.iTyp * 1000000) + T_Station.THardware.TAxisToolCenter.T_CtrleSingle.udiErrorID;
				ELSE
					diErrorNr:=0;
				END_IF;
			END_IF;
			IF T_Station.THardware.TAxisToolFeeder.T_CtrleSingle.xErr AND NOT(xMicroRodActive) THEN
				IF (T_Station.THardware.TAxisToolFeeder.T_Config_Gen.iTyp <> 0) THEN
					diErrorNr:=(T_Station.THardware.TAxisToolFeeder.T_Config_Gen.iTyp * 1000000) + T_Station.THardware.TAxisToolFeeder.T_CtrleSingle.udiErrorID;
				ELSE
					diErrorNr:=0;
				END_IF;
			END_IF;
			FBErrorMessage(	diErrorNr:=diErrorNr,
							T_ErrorList:=T_ErrorList);
			T_Visu.ptrT_ExchgParam^.T_Visu.T_Message.sDynamicTextEnglish:=FBErrorMessage.sErrorTextEnglish;
			T_Visu.ptrT_ExchgParam^.T_Visu.T_Message.sDynamicTextDeutsch:=FBErrorMessage.sErrorTextDeutsch;
			T_Visu.ptrT_ExchgParam^.T_Visu.T_Message.sDynamicTextFrancais:=FBErrorMessage.sErrorTextFrancais;
			T_Visu.ptrT_ExchgParam^.T_SafetyCtrl.xSetForceError:=TRUE;
			T_Visu.ptrT_ExchgParam^.T_SafetyCtrl.diSetForceErrorNr:=diErrorNr;
			T_Visu.T_CtrleAction.xErr:=FALSE;
			T_Visu.T_CtrleAction.udiErrorID:=0;
			T_Station.THardware.TAxisToolRight.T_CtrleSingle.iFunction:=1;
			T_Station.THardware.TAxisToolCenter.T_CtrleSingle.iFunction:=1;
			T_Station.THardware.TAxisToolFeeder.T_CtrleSingle.iFunction:=1;
			T_Station.THardware.TAxisToolRight.T_CtrleSingle.xExecute:=T_Station.THardware.TAxisToolRight.T_CtrleSingle.xErr;
			T_Station.THardware.TAxisToolCenter.T_CtrleSingle.xExecute:=T_Station.THardware.TAxisToolCenter.T_CtrleSingle.xErr AND xMicroRodActive;
			T_Station.THardware.TAxisToolFeeder.T_CtrleSingle.xExecute:=T_Station.THardware.TAxisToolFeeder.T_CtrleSingle.xErr AND NOT(xMicroRodActive);
			xSwitchMasterSlave:=FALSE;
		END_CASE
	END_IF;

(* Action cylinder toggle state *)
	IF xToggleCylinderState THEN
		(* Step toggle state *)
		CASE iStepAction OF
		(* check cylinder state *)
		1:	xTmp:=	ptrCylAction^.T_CtrleCyl.xDone
					AND NOT(ptrCylAction^.T_CtrleCyl.xExecute)
					AND NOT(ptrCylAction^.T_CtrleCyl.xErr);
			(* next step *)
			IF xTmp THEN iStepAction:=10; ELSE iStepAction:=95; END_IF
			IF xTmp AND T_Station.TControl.xHardwareConfigError THEN iStepAction:=95; END_IF;
		(* toggle cylinder state *)
		10:	ptrCylAction^.T_CtrleCyl.iFunction:=51;
			ptrCylAction^.T_CtrleCyl.xExecute:=TRUE;
			(* next step *)
			iStepAction:=20;
			xStepActionDone:=FALSE;
		(* wait confirmation *)
		20:	IF NOT(xStepActionDone) THEN
			(* release execution *)
				ptrCylAction^.T_CtrleCyl.xExecute:=FALSE;
				xStepActionDone:=TRUE;
			ELSE
				IF ptrCylAction^.T_CtrleCyl.xDone THEN
				(* action done *)
					iStepAction:=90;
					xStepActionDone:=FALSE;
				ELSE 	IF ptrCylAction^.T_CtrleCyl.xErr THEN
						(* action error *)
							iStepAction:=99;
							xStepActionDone:=FALSE;
						END_IF
				END_IF
			END_IF
		(* waiting time out *)
		89:	IF TimerAction.Q THEN iStepAction:=90; END_IF
		(* action done *)
		90:	T_Visu.T_CtrleAction.xDone:=TRUE;
			T_Visu.T_CtrleAction.xNotReady:=FALSE;
			T_Visu.T_CtrleAction.xErr:=FALSE;
			T_Visu.T_CtrleAction.udiErrorID:=0;
			xToggleCylinderState:=FALSE;
		(* cylinder not ready *)
		95:	TimerNotReady(IN:=TRUE);
			xToggleCylinderState:=FALSE;
		(* error *)
		99:	T_Visu.T_CtrleAction.xDone:=TRUE;
			T_Visu.T_CtrleAction.xNotReady:=FALSE;
			(*diErrorNr:=6000000 * ptrCylAction^.T_CtrleCyl.udiErrorID;*)
			diErrorNr:=9000000+ (1000000 * iSelectedCylinder) + ptrCylAction^.T_CtrleCyl.udiErrorID;
			FBErrorMessage(	diErrorNr:=diErrorNr,
							T_ErrorList:=T_ErrorList);
			T_Visu.ptrT_ExchgParam^.T_Visu.T_Message.sDynamicTextEnglish:=FBErrorMessage.sErrorTextEnglish;
			T_Visu.ptrT_ExchgParam^.T_Visu.T_Message.sDynamicTextDeutsch:=FBErrorMessage.sErrorTextDeutsch;
			T_Visu.ptrT_ExchgParam^.T_Visu.T_Message.sDynamicTextFrancais:=FBErrorMessage.sErrorTextFrancais;
			T_Visu.ptrT_ExchgParam^.T_SafetyCtrl.xSetForceError:=TRUE;
			T_Visu.ptrT_ExchgParam^.T_SafetyCtrl.diSetForceErrorNr:=diErrorNr;
			T_Visu.T_CtrleAction.xErr:=FALSE;
			T_Visu.T_CtrleAction.udiErrorID:=0;
			ptrCylAction^.T_CtrleCyl.xReset:=TRUE;
			xToggleCylinderState:=FALSE;
		END_CASE
	END_IF

(* ToolTens force +,++,-,-- *)
	IF xToolTensForceAdd OR xToolTensForceAddMore OR xToolTensForceSub OR xToolTensForceSubMore THEN
		CASE iStepAction OF
		(* check cylinder state *)
		1:	xTmp:=	ptrCylAction^.T_CtrleCyl.xDone
					AND NOT(ptrCylAction^.T_CtrleCyl.xExecute)
					AND NOT(ptrCylAction^.T_CtrleCyl.xErr)
					AND ptrCylAction^.T_CtrleCyl.T_AnalogCylinder.xActiv;
			(* next step *)
			IF xTmp THEN iStepAction:=10; ELSE iStepAction:=95; END_IF
			IF xTmp AND T_Station.TControl.xHardwareConfigError THEN iStepAction:=95; END_IF;
		10:	IF xToolTensForceAdd THEN
				rCorrectionValue:=0.1;
			END_IF;
			IF xToolTensForceAddMore THEN
				rCorrectionValue:=1.0;
			END_IF;
			IF xToolTensForceSub THEN
				rCorrectionValue:=-0.1;
			END_IF;
			IF xToolTensForceSubMore THEN
				rCorrectionValue:=-1.0;
			END_IF;
			T_Visu.ptrT_ExchgParam^.T_InfoValueCommon.rToolTensionForce:=T_Visu.ptrT_ExchgParam^.T_InfoValueCommon.rToolTensionForce + rCorrectionValue;
			IF (T_Visu.ptrT_ExchgParam^.T_InfoValueCommon.rToolTensionForce < 0.1) THEN
				T_Visu.ptrT_ExchgParam^.T_InfoValueCommon.rToolTensionForce:=0.0;
			END_IF;
			IF (T_Visu.ptrT_ExchgParam^.T_InfoValueCommon.rToolTensionForce > T_NovRAM.T_Data.T_Standard.T_ToolTensionSystem.rMaxForceTT) THEN
				T_Visu.ptrT_ExchgParam^.T_InfoValueCommon.rToolTensionForce:=T_NovRAM.T_Data.T_Standard.T_ToolTensionSystem.rMaxForceTT;
			END_IF;
			(* next step *)
			iStepAction:=20;
		(* activ function set analog value *)
		20:	ptrCylAction^.T_CtrleCyl.T_AnalogCylinder.rForceIn:=T_Visu.ptrT_ExchgParam^.T_InfoValueCommon.rToolTensionForce;
			ptrCylAction^.T_CtrleCyl.iFunction:=4;
			ptrCylAction^.T_CtrleCyl.xExecute:=TRUE;
			(* next step *)
			iStepAction:=30;
			xStepActionDone:=FALSE;
		(* wait confirmation *)
		30:	IF NOT(xStepActionDone) THEN
			(* release execution *)
				ptrCylAction^.T_CtrleCyl.xExecute:=FALSE;
				xStepActionDone:=TRUE;
			ELSE
				IF ptrCylAction^.T_CtrleCyl.xDone THEN
				(* action done *)
					iStepAction:=90;
					xStepActionDone:=FALSE;
				ELSE 	IF ptrCylAction^.T_CtrleCyl.xErr THEN
						(* action error *)
							iStepAction:=99;
							xStepActionDone:=FALSE;
						END_IF
				END_IF
			END_IF
		(* waiting time out *)
		89:	IF TimerAction.Q THEN iStepAction:=90; END_IF
		(* action done *)
		90:	T_Visu.T_CtrleAction.xDone:=TRUE;
			T_Visu.T_CtrleAction.xNotReady:=FALSE;
			T_Visu.T_CtrleAction.xErr:=FALSE;
			T_Visu.T_CtrleAction.udiErrorID:=0;
			xToolTensForceAdd:=xToolTensForceAddMore:=xToolTensForceSub:=xToolTensForceSubMore:=FALSE;
		(* cylinder not ready *)
		95:	TimerNotReady(IN:=TRUE);
			xToolTensForceAdd:=xToolTensForceAddMore:=xToolTensForceSub:=xToolTensForceSubMore:=FALSE;
		(* error *)
		99:	T_Visu.T_CtrleAction.xDone:=TRUE;
			T_Visu.T_CtrleAction.xNotReady:=FALSE;
			(*diErrorNr:=6000000 * ptrCylAction^.T_CtrleCyl.udiErrorID;*)
			diErrorNr:=9000000+ (1000000 * iSelectedCylinder) + ptrCylAction^.T_CtrleCyl.udiErrorID;
			FBErrorMessage(	diErrorNr:=diErrorNr,
							T_ErrorList:=T_ErrorList);
			T_Visu.ptrT_ExchgParam^.T_Visu.T_Message.sDynamicTextEnglish:=FBErrorMessage.sErrorTextEnglish;
			T_Visu.ptrT_ExchgParam^.T_Visu.T_Message.sDynamicTextDeutsch:=FBErrorMessage.sErrorTextDeutsch;
			T_Visu.ptrT_ExchgParam^.T_Visu.T_Message.sDynamicTextFrancais:=FBErrorMessage.sErrorTextFrancais;
			T_Visu.ptrT_ExchgParam^.T_SafetyCtrl.xSetForceError:=TRUE;
			T_Visu.ptrT_ExchgParam^.T_SafetyCtrl.diSetForceErrorNr:=diErrorNr;
			T_Visu.T_CtrleAction.xErr:=FALSE;
			T_Visu.T_CtrleAction.udiErrorID:=0;
			ptrCylAction^.T_CtrleCyl.xReset:=TRUE;
			xToolTensForceAdd:=xToolTensForceAddMore:=xToolTensForceSub:=xToolTensForceSubMore:=FALSE;
		END_CASE
	END_IF;

(* Action Station Function *)
	IF xActivateStationFunction THEN;
		(* Step  function station  *)
		CASE iStepAction OF
		(* check station state *)
		1:	xTmp:=	T_Station.TControl.xEnd AND
					T_Station.TControl.xRdy AND
					NOT(T_Station.TControl.xStart) AND
					NOT(T_Station.TControl.xError) AND
					NOT(T_Station.TControl.xStop) AND
					( (T_Visu.ptrT_ExchgParam^.T_StationCommon.rNewToolRotationSpeed <> 0) OR (iTmpStationFunctionNr = 20)) ;
			(* next step *)
			IF xTmp THEN iStepAction:=20; ELSE iStepAction:=95; END_IF
			IF xTmp AND T_Station.TControl.xHardwareConfigError THEN iStepAction:=95; END_IF;
		(* determin function number *)
		20:	IF (iTmpStationFunctionNr = 2) THEN
				bStateMachine:=2;
				xSetStateMachine:=TRUE;
			END_IF;
			T_Station.TControl.iFunctNr:=iTmpStationFunctionNr;
			CASE T_Station.TControl.iFunctNr OF
			(* available function, activ function *)
			2,3:	CASE T_Station.TControl.iFunctNr OF
				2:	T_Station.THardware.TAxisToolLeft.T_CtrleSingle.lrVelocity:=T_Visu.ptrT_ExchgParam^.T_StationCommon.rNewToolRotationSpeed;
					T_Station.THardware.TAxisToolLeft.T_CtrleSingle.lrAcceleration:=T_NovRAM.T_Data.T_Standard.T_TeachINToolLeft.rAcceleration;
					T_Station.THardware.TAxisToolLeft.T_CtrleSingle.lrDecceleration:=T_NovRAM.T_Data.T_Standard.T_TeachINToolLeft.rDeceleration;
					T_Station.THardware.TAxisToolLeft.T_CtrleSingle.lrGearDivider:=10000;
					T_Station.THardware.TAxisToolLeft.T_CtrleSingle.lrGearFactor:=10000;

					IF xMicroRodActive THEN
						(* ToolCenter --> Slave of ToolLeft only by MicroRod *)
						T_Station.THardware.TAxisToolCenter.T_CtrleSingle.lrAcceleration:=T_NovRAM.T_Data.T_Standard.T_TeachINToolCenter.rAcceleration;
						T_Station.THardware.TAxisToolCenter.T_CtrleSingle.lrDecceleration:=T_NovRAM.T_Data.T_Standard.T_TeachINToolCenter.rDeceleration;
						T_Station.THardware.TAxisToolCenter.T_CtrleSingle.lrGearDivider:=INT_TO_LREAL(T_Station.T_WorkTool.iBaseGearDivider);
						T_Station.THardware.TAxisToolCenter.T_CtrleSingle.lrGearFactor:=(	INT_TO_LREAL(T_Station.T_WorkTool.iBaseGearDivider) /
																						(T_Station.THardware.TAxisToolLeft.T_CtrleSingle.lrGearRatio /
																						T_Station.THardware.TAxisToolCenter.T_CtrleSingle.lrGearRatio)) * -1.0;
						(* ToolRight --> Slave of ToolLeft by MicroWire or Slave of ToolRight by MicroRod *)
						T_Station.THardware.TAxisToolRight.T_CtrleSingle.lrAcceleration:=T_NovRAM.T_Data.T_Standard.T_TeachINToolRight.rAcceleration;
						T_Station.THardware.TAxisToolRight.T_CtrleSingle.lrDecceleration:=T_NovRAM.T_Data.T_Standard.T_TeachINToolRight.rDeceleration;
						T_Station.THardware.TAxisToolRight.T_CtrleSingle.lrGearDivider:=INT_TO_LREAL(T_Station.T_WorkTool.iBaseGearDivider);
						T_Station.THardware.TAxisToolRight.T_CtrleSingle.lrGearFactor:=	INT_TO_LREAL(T_Station.T_WorkTool.iBaseGearDivider) /
																						(T_Station.THardware.TAxisToolLeft.T_CtrleSingle.lrGearRatio /
																						T_Station.THardware.TAxisToolRight.T_CtrleSingle.lrGearRatio);
					END_IF;
					IF NOT(xMicroRodActive) THEN
						(* ToolRight --> Slave of ToolRight by MicroWire *)
						T_Station.THardware.TAxisToolFeeder.T_CtrleSingle.lrAcceleration:=T_NovRAM.T_Data.T_Standard.T_TeachINToolFeeder.rAcceleration;
						T_Station.THardware.TAxisToolFeeder.T_CtrleSingle.lrDecceleration:=T_NovRAM.T_Data.T_Standard.T_TeachINToolFeeder.rDeceleration;
						T_Station.THardware.TAxisToolFeeder.T_CtrleSingle.lrGearDivider:=INT_TO_LREAL(T_Station.T_WorkTool.iBaseGearDivider);
						T_Station.THardware.TAxisToolFeeder.T_CtrleSingle.lrGearFactor:=	(INT_TO_LREAL(T_Station.T_WorkTool.iBaseGearDivider) /
																						(T_Station.THardware.TAxisToolFeeder.T_CtrleSingle.lrGearRatio /
																						T_Station.THardware.TAxisToolRight.T_CtrleSingle.lrGearRatio)) * -1.0;

						(* ToolRight --> Slave of ToolLeft by MicroWire or Slave of ToolRight by MicroRod *)
						T_Station.THardware.TAxisToolRight.T_CtrleSingle.lrAcceleration:=T_NovRAM.T_Data.T_Standard.T_TeachINToolRight.rAcceleration;
						T_Station.THardware.TAxisToolRight.T_CtrleSingle.lrDecceleration:=T_NovRAM.T_Data.T_Standard.T_TeachINToolRight.rDeceleration;
						T_Station.THardware.TAxisToolRight.T_CtrleSingle.lrGearDivider:=INT_TO_LREAL(T_Station.T_WorkTool.iBaseGearDivider);
						T_Station.THardware.TAxisToolRight.T_CtrleSingle.lrGearFactor:=	(INT_TO_LREAL(T_Station.T_WorkTool.iBaseGearDivider) /
																						(T_Station.THardware.TAxisToolLeft.T_CtrleSingle.lrGearRatio /
																						T_Station.THardware.TAxisToolRight.T_CtrleSingle.lrGearRatio)) * -1.0;
					END_IF;
				END_CASE;
				T_Station.TControl.xStart:=TRUE;
				IF (T_Station.TControl.iFunctNr = 2) THEN
					(* Display message *)
					T_Visu.ptrT_ExchgParam^.T_Visu.T_Message.iState:=25;
				END_IF;
				(* next step *)
				iStepAction:=30;
			(* not available function *)
			20:	T_Station.TControl.xStart:=TRUE;
			T_Visu.ptrT_ExchgParam^.T_Visu.T_Message.iState:=2;
(*				T_Visu.ptrT_ExchgParam^.T_SafetyCtrl.bStateReferenceMaxToolLength:=2;*)
				bStateMachine:=2;
				xSetStateMachine:=TRUE;
			    	iStepAction:=30;
			1,4..19,21..99:		iStepAction:=95;
			END_CASE
			(* next step *)
			xStepActionDone:=FALSE;
		(* wait confirmation *)
		30:	IF NOT(xStepActionDone) THEN
			(* release execution *)
				T_Station.TControl.xStart:=FALSE;
				xStepActionDone:=TRUE;
			ELSE
				IF T_Station.TControl.xEnd THEN
				(* action done *)
					IF(iTmpStationFunctionNr = 20) THEN
						iStepAction:=50;
					ELSE
						iStepAction:=90;
					END_IF;
					xStepActionDone:=FALSE;
				ELSE 	IF T_Station.TControl.xError THEN
						(* action error *)
							iStepAction:=99;
							xStepActionDone:=FALSE;
						END_IF
				END_IF
			END_IF
		(* Save NovRam *)
		50:	T_NovRam.T_Data.T_Standard.T_MachineConfig.rConfigMaxToolLength:=T_Station.THardware.TAxisToolFeeder.T_LiveValue.lrActualPosition *0.1;
			T_NovRam.T_Data.T_Standard.T_MachineConfig.rConfigMaxToolLengthOriginal:=T_Station.THardware.TAxisToolFeeder.T_LiveValue.lrActualPosition *0.1;
			T_Station.xOverwriteMaxToolLength:=TRUE;
			T_NovRAM.T_Ctrle.xExecute:=TRUE;
			T_NovRAM.T_Ctrle.iFunction:=2;
			iStepAction:=60;
		60:	IF NOT(xStepActionDone) THEN
				xStepActionDone:=TRUE;
				T_NovRAM.T_Ctrle.xExecute:=FALSE;
			END_IF;
			IF T_NovRAM.T_Ctrle.xDone THEN
				T_Station.T_MachineConfig.rConfigMaxToolLength:=T_NovRAM.T_Data.T_Standard.T_MachineConfig.rConfigMaxToolLength;
				T_Station.xOverwriteMaxToolLength:=FALSE;
				xStepActionDone:=FALSE;
				iStepAction:=90;
			END_IF;
		(* action done *)
		90:	IF (iTmpStationFunctionNr = 3) THEN
				bStateMachine:=1;
				xSetStateMachine:=TRUE;
			END_IF;
			IF (iTmpStationFunctionNr = 20) THEN
				T_Visu.ptrT_ExchgParam^.T_StationCommon.rConfigMaxToolLength:=T_NovRAM.T_Data.T_Standard.T_MachineConfig.rConfigMaxToolLength;
				T_Visu.ptrT_ExchgParam^.T_StationCommon.rConfigMaxToolLengthOriginal:=T_NovRAM.T_Data.T_Standard.T_MachineConfig.rConfigMaxToolLength;
				T_Visu.ptrT_ExchgParam^.T_Visu.T_Message.iState:=1;
(*				T_Visu.ptrT_ExchgParam^.T_SafetyCtrl.bStateReferenceMaxToolLength:=1;*)
				bStateMachine:=1;
				xSetStateMachine:=TRUE;
			END_IF;
			T_Visu.T_CtrleAction.xDone:=TRUE;
			T_Visu.T_CtrleAction.xNotReady:=FALSE;
			T_Visu.T_CtrleAction.xErr:=FALSE;
			T_Visu.T_CtrleAction.udiErrorID:=0;
			xActivateStationFunction:=FALSE;
		(* Configuration Error *)
		91:	T_Visu.T_CtrleAction.xDone:=TRUE;
			T_Visu.T_CtrleAction.xNotReady:=FALSE;
			T_Visu.T_CtrleAction.xErr:=FALSE;
			T_Visu.T_CtrleAction.udiErrorID:=0;
			xActivateStationFunction:=FALSE;
		(* function not ready *)
		95:	TimerNotReady(IN:=TRUE);
			xActivateStationFunction:=FALSE;
		(* error *)
		99:	T_Visu.T_CtrleAction.xDone:=TRUE;
			T_Visu.T_CtrleAction.xNotReady:=FALSE;
			FBErrorMessage(	diErrorNr:=T_Station.TControl.diErrorNr,
							T_ErrorList:=T_ErrorList);
			T_Visu.ptrT_ExchgParam^.T_Visu.T_Message.sDynamicTextEnglish:=FBErrorMessage.sErrorTextEnglish;
			T_Visu.ptrT_ExchgParam^.T_Visu.T_Message.sDynamicTextDeutsch:=FBErrorMessage.sErrorTextDeutsch;
			T_Visu.ptrT_ExchgParam^.T_Visu.T_Message.sDynamicTextFrancais:=FBErrorMessage.sErrorTextFrancais;
			T_Visu.T_CtrleAction.xErr:=FALSE;
			T_Visu.T_CtrleAction.udiErrorID:=0;
			xActivateStationFunction:=FALSE;
		END_CASE
	END_IF;

(* Activation of the Section for the ToolGeometry *)
	IF xActivationSection1 OR xActivationSection2 OR xActivationSection3 OR xActivationSection4 OR xActivationSection5 OR xActivationSection6 OR xSetPitchEqual THEN
		CASE iStepAction OF
		(* check visu *)
		1:	xTmp:=	TRUE;
			IF xTmp THEN
				(* next Step *)
				iStepAction :=10;
			(* activ error *)
			ELSE iStepAction:=95; END_IF
		(* Set parameter page *)
		10:	ptxActiveSection1:=ADR(T_Visu.ptrT_ExchgParam^.T_GeometryCommon.T_Geometry.axActiveSection[1]);
			ptxActiveSection2:=ADR(T_Visu.ptrT_ExchgParam^.T_GeometryCommon.T_Geometry.axActiveSection[2]);
			ptxActiveSection3:=ADR(T_Visu.ptrT_ExchgParam^.T_GeometryCommon.T_Geometry.axActiveSection[3]);
			ptxActiveSection4:=ADR(T_Visu.ptrT_ExchgParam^.T_GeometryCommon.T_Geometry.axActiveSection[4]);
			ptxActiveSection5:=ADR(T_Visu.ptrT_ExchgParam^.T_GeometryCommon.T_Geometry.axActiveSection[5]);
			ptxActiveSection6:=ADR(T_Visu.ptrT_ExchgParam^.T_GeometryCommon.T_Geometry.axActiveSection[6]);

(*** Checking if: the section is already active / is the olny active / a section before is active  ***)
			IF xActivationSection1 THEN
				IF (ptxActiveSection1^ AND NOT(ptxActiveSection2^)) OR
				     (NOT(ptxActiveSection1^) AND NOT(ptxActiveSection2^) AND (ptxActiveSection3^ OR ptxActiveSection4^OR ptxActiveSection5^ OR ptxActiveSection6^)) THEN
					;
				ELSE
					ptxActiveSection1^:=NOT(ptxActiveSection1^);
				END_IF;
			END_IF;

			IF xActivationSection2 THEN
				IF (ptxActiveSection2^ AND ptxActiveSection1^ AND ptxActiveSection3^) OR
				    (ptxActiveSection2^ AND NOT(ptxActiveSection1^) AND NOT(ptxActiveSection3^)) OR
				    (NOT(ptxActiveSection2^) AND NOT(ptxActiveSection1^) AND NOT(ptxActiveSection3^) AND (ptxActiveSection4^OR ptxActiveSection5^ OR ptxActiveSection6^)) THEN
					;
				ELSE
					ptxActiveSection2^:=NOT(ptxActiveSection2^);
				END_IF;
			END_IF;
				IF xActivationSection3 THEN
					IF (ptxActiveSection3^ AND ptxActiveSection2^ AND ptxActiveSection4^) OR
					    (ptxActiveSection3^ AND NOT(ptxActiveSection2^) AND NOT(ptxActiveSection4^)) OR
					    (NOT(ptxActiveSection3^) AND NOT(ptxActiveSection2^) AND NOT(ptxActiveSection4^) AND (ptxActiveSection5^ OR ptxActiveSection6^ OR ptxActiveSection1^))THEN
						;
					ELSE
						ptxActiveSection3^:=NOT(ptxActiveSection3^);
					END_IF;
				END_IF;
			IF xActivationSection4 THEN
				IF (ptxActiveSection4^ AND ptxActiveSection3^ AND ptxActiveSection5^) OR
				    (ptxActiveSection4^ AND NOT(ptxActiveSection3^) AND NOT(ptxActiveSection5^)) OR
				    (NOT(ptxActiveSection4^) AND NOT(ptxActiveSection3^) AND NOT(ptxActiveSection5^) AND (ptxActiveSection6^OR ptxActiveSection1^ OR ptxActiveSection2^)) THEN
					;
				ELSE
					ptxActiveSection4^:=NOT(ptxActiveSection4^);
				END_IF;
			END_IF;
(*09.12.2022: SOA	{	 *)
				IF xActivationSection5 THEN
					IF (ptxActiveSection5^ AND ptxActiveSection4^ AND ptxActiveSection6^) OR
					    (ptxActiveSection5^ AND NOT(ptxActiveSection4^) AND NOT(ptxActiveSection6^)) OR
					    (NOT(ptxActiveSection5^) AND NOT(ptxActiveSection4^) AND NOT(ptxActiveSection6^) AND (ptxActiveSection1^ OR ptxActiveSection2^ OR ptxActiveSection3^))THEN
						;
					ELSE
						ptxActiveSection5^:=NOT(ptxActiveSection5^);
					END_IF;
				END_IF;
			IF xActivationSection6 THEN
				IF (ptxActiveSection6^ AND NOT(ptxActiveSection5^)) OR
				    (NOT(ptxActiveSection6^) AND NOT(ptxActiveSection5^) AND (ptxActiveSection1^ OR ptxActiveSection2^ OR ptxActiveSection3^ OR ptxActiveSection4^ )) THEN
					;
				ELSE
					ptxActiveSection6^:=NOT(ptxActiveSection6^);
				END_IF;
			END_IF;
(*09.12.2022: SOA	}	 *)
(*09.12.2022: SOA	{	 *)
			IF xSetPitchEqual THEN
				IF T_Visu.ptrT_ExchgParam^.T_GeometryCommon.T_Geometry.axActiveSection[1] THEN
					rSectionPitch:=T_Visu.ptrT_ExchgParam^.T_GeometryCommon.T_Geometry.arSectionPitch[1];
					IF T_Visu.ptrT_ExchgParam^.T_GeometryCommon.T_Geometry.axActiveSection[2] THEN
						T_Visu.ptrT_ExchgParam^.T_GeometryCommon.T_Geometry.arSectionPitch[2]:=rSectionPitch;
					END_IF;
					IF T_Visu.ptrT_ExchgParam^.T_GeometryCommon.T_Geometry.axActiveSection[3] THEN
						T_Visu.ptrT_ExchgParam^.T_GeometryCommon.T_Geometry.arSectionPitch[3]:=rSectionPitch;
					END_IF;
					IF T_Visu.ptrT_ExchgParam^.T_GeometryCommon.T_Geometry.axActiveSection[4] THEN
						T_Visu.ptrT_ExchgParam^.T_GeometryCommon.T_Geometry.arSectionPitch[4]:=rSectionPitch;
					END_IF;
					IF T_Visu.ptrT_ExchgParam^.T_GeometryCommon.T_Geometry.axActiveSection[5] THEN
						T_Visu.ptrT_ExchgParam^.T_GeometryCommon.T_Geometry.arSectionPitch[5]:=rSectionPitch;
					END_IF;
					IF T_Visu.ptrT_ExchgParam^.T_GeometryCommon.T_Geometry.axActiveSection[6] THEN
						T_Visu.ptrT_ExchgParam^.T_GeometryCommon.T_Geometry.arSectionPitch[6]:=rSectionPitch;
					END_IF;
				ELSIF T_Visu.ptrT_ExchgParam^.T_GeometryCommon.T_Geometry.axActiveSection[2] THEN
					rSectionPitch:=T_Visu.ptrT_ExchgParam^.T_GeometryCommon.T_Geometry.arSectionPitch[2];
					IF T_Visu.ptrT_ExchgParam^.T_GeometryCommon.T_Geometry.axActiveSection[3] THEN
						T_Visu.ptrT_ExchgParam^.T_GeometryCommon.T_Geometry.arSectionPitch[3]:=rSectionPitch;
					END_IF;
					IF T_Visu.ptrT_ExchgParam^.T_GeometryCommon.T_Geometry.axActiveSection[4] THEN
						T_Visu.ptrT_ExchgParam^.T_GeometryCommon.T_Geometry.arSectionPitch[4]:=rSectionPitch;
					END_IF;
					IF T_Visu.ptrT_ExchgParam^.T_GeometryCommon.T_Geometry.axActiveSection[5] THEN
						T_Visu.ptrT_ExchgParam^.T_GeometryCommon.T_Geometry.arSectionPitch[5]:=rSectionPitch;
					END_IF;
					IF T_Visu.ptrT_ExchgParam^.T_GeometryCommon.T_Geometry.axActiveSection[6] THEN
						T_Visu.ptrT_ExchgParam^.T_GeometryCommon.T_Geometry.arSectionPitch[6]:=rSectionPitch;
					END_IF;
				ELSIF T_Visu.ptrT_ExchgParam^.T_GeometryCommon.T_Geometry.axActiveSection[3] THEN
					rSectionPitch:=T_Visu.ptrT_ExchgParam^.T_GeometryCommon.T_Geometry.arSectionPitch[3];
					IF T_Visu.ptrT_ExchgParam^.T_GeometryCommon.T_Geometry.axActiveSection[4] THEN
						T_Visu.ptrT_ExchgParam^.T_GeometryCommon.T_Geometry.arSectionPitch[4]:=rSectionPitch;
					END_IF;
					IF T_Visu.ptrT_ExchgParam^.T_GeometryCommon.T_Geometry.axActiveSection[5] THEN
						T_Visu.ptrT_ExchgParam^.T_GeometryCommon.T_Geometry.arSectionPitch[5]:=rSectionPitch;
					END_IF;
					IF T_Visu.ptrT_ExchgParam^.T_GeometryCommon.T_Geometry.axActiveSection[6] THEN
						T_Visu.ptrT_ExchgParam^.T_GeometryCommon.T_Geometry.arSectionPitch[6]:=rSectionPitch;
					END_IF;
				ELSIF T_Visu.ptrT_ExchgParam^.T_GeometryCommon.T_Geometry.axActiveSection[4] THEN
					rSectionPitch:=T_Visu.ptrT_ExchgParam^.T_GeometryCommon.T_Geometry.arSectionPitch[4];
					IF T_Visu.ptrT_ExchgParam^.T_GeometryCommon.T_Geometry.axActiveSection[5] THEN
						T_Visu.ptrT_ExchgParam^.T_GeometryCommon.T_Geometry.arSectionPitch[5]:=rSectionPitch;
					END_IF;
					IF T_Visu.ptrT_ExchgParam^.T_GeometryCommon.T_Geometry.axActiveSection[6] THEN
						T_Visu.ptrT_ExchgParam^.T_GeometryCommon.T_Geometry.arSectionPitch[6]:=rSectionPitch;
					END_IF;
				ELSIF T_Visu.ptrT_ExchgParam^.T_GeometryCommon.T_Geometry.axActiveSection[5] THEN
					rSectionPitch:=T_Visu.ptrT_ExchgParam^.T_GeometryCommon.T_Geometry.arSectionPitch[5];
					IF T_Visu.ptrT_ExchgParam^.T_GeometryCommon.T_Geometry.axActiveSection[6] THEN
						T_Visu.ptrT_ExchgParam^.T_GeometryCommon.T_Geometry.arSectionPitch[6]:=rSectionPitch;
					END_IF;
				ELSIF T_Visu.ptrT_ExchgParam^.T_GeometryCommon.T_Geometry.axActiveSection[6] THEN
					rSectionPitch:=T_Visu.ptrT_ExchgParam^.T_GeometryCommon.T_Geometry.arSectionPitch[6];
				END_IF;
			END_IF;
(*09.12.2022: SOA	}   *)
			iStepAction :=90;
		(* change page done *)
		90:	T_Visu.T_CtrleAction.xDone:=TRUE;
			T_Visu.T_CtrleAction.xNotReady:=FALSE;
			T_Visu.T_CtrleAction.xErr:=FALSE;
			T_Visu.T_CtrleAction.udiErrorID:=0;
			xActivationSection1:=xActivationSection2:=xActivationSection3:=xActivationSection4:=xActivationSection5:=xActivationSection6:=xSetPitchEqual:=FALSE;
		(* not ready *)
		95:	T_Visu.T_CtrleAction.xDone:=TRUE;
			T_Visu.T_CtrleAction.xNotReady:=FALSE;
			T_Visu.T_CtrleAction.xErr:=FALSE;
			T_Visu.T_CtrleAction.udiErrorID:=0;
			xActivationSection1:=xActivationSection2:=xActivationSection3:=xActivationSection4:=xActivationSection5:=xActivationSection6:=xSetPitchEqual:=FALSE;
		(* error *)
		99:	T_Visu.T_CtrleAction.xDone:=FALSE;
			T_Visu.T_CtrleAction.xNotReady:=FALSE;
			T_Visu.T_CtrleAction.xErr:=TRUE;
			T_Visu.T_CtrleAction.udiErrorID:=16#F0000 + T_Visu.T_CtrleAction.iFunction;
			xActivationSection1:=xActivationSection2:=xActivationSection3:=xActivationSection4:=xActivationSection5:=xActivationSection6:=xSetPitchEqual:=FALSE;
		END_CASE
	END_IF;


(* Copy profile value to process *)
	IF xAction_CopyProfileToProcess THEN
		(* Set copy action *)
		CASE iStepAction OF
		(* Set default value *)
		1:	(*IF xFctSetDefaultValueProfileOnlineChange(ptrNovRAM:=ADR(T_WorkingData),
												   ptrDefaultProfilStandProcPara:=ADR(T_DefaultProfilStandProcPara),
												   bActiveStation:=0) THEN iStepAction:=5; END_IF*)
			iStepAction:=10;
			(* Init. display value *)
			xProfileFileNotFound:=FALSE;
		(* activ reading profile file *)
		10:	IF (T_Visu.ptrT_ExchgParam^.T_StationCommon.T_InfoProcess.iProfile > 0) AND (T_Visu.ptrT_ExchgParam^.T_StationCommon.T_InfoProcess.iProfile <= csiMaxProfile) THEN
				T_Profile.T_Id.iNumber:=T_Visu.ptrT_ExchgParam^.T_StationCommon.T_InfoProcess.iProfile;
				T_Profile.T_Id.sName:=T_Visu.ptrT_ExchgParam^.T_StationCommon.T_InfoProcess.sProfileName;
				T_Profile.T_Ctrle.iFunction:=1;
				T_Profile.T_Ctrle.xExecute:=TRUE;
				(* next step *)
				iStepAction:=20;
			ELSE iStepAction:=25; END_IF
		20:	IF NOT T_Profile.T_Ctrle.xExecute AND T_Profile.T_Ctrle.xDone THEN
				(* next step *)
				iStepAction:=90;
			END_IF
			IF T_Profile.T_Ctrle.xErr THEN
				xProfileFileNotFound:=TRUE;
				iToLoadProfileNr:=T_Profile.T_Id.iNumber;
				sToLoadProfileName:=T_Profile.T_Id.sName;
				(* activ reset *)
				T_Profile.T_Ctrle.xReset:=TRUE;
				(* next step *)
				iStepAction:=25;
			END_IF
		(* waiting flag *)
		25:	IF NOT T_Profile.T_Ctrle.xReset AND T_Profile.T_Ctrle.xDone THEN
				IF (T_Profile.T_Id.iNumber = 1) THEN
					(*T_ActualProfilStandProcPara[1]:=T_DefaultProfilStandProcPara[1];*)
					iStepAction:=90;
				ELSE
					iStepAction:=26;
				END_IF;
				(* erase name *)
				T_NovRam.T_Data.T_IDProfileStation[1].sName:='Default';
				T_NovRam.T_Data.T_IDProfileStation[1].iNumber:=1;
				T_Visu.ptrT_ExchgParam^.T_StationCommon.T_InfoProcess.sProfileName:='Default';
				T_Visu.ptrT_ExchgParam^.T_StationCommon.T_InfoProcess.iProfile:=1;
			END_IF
			IF T_Profile.T_Ctrle.xErr THEN iStepAction:=99; END_IF
		(* activ reading profile file *)
		26:	T_Profile.T_Id.iNumber:=1;
			T_Profile.T_Id.sName:='Default';
			T_Profile.T_Ctrle.iFunction:=1;
			T_Profile.T_Ctrle.xExecute:=TRUE;
			(* next step *)
			iStepAction:=20;
		(* End function *)
		90:	IF xProfileFileNotFound THEN
				xProfileFileNotFound:=FALSE;
				sTmpDynamicText:=INT_TO_STRING(iToLoadProfileNr);
				sTmpDynamicText:=CONCAT(sTmpDynamicText,' ');
				(* For English Language *)
				T_Visu.ptrT_ExchgParam^.T_Visu.T_Message.sDynamicTextEnglish:=CONCAT(T_ErrorList.asErrorListEnglish.T_LanguagList[50],sTmpDynamicText);	(* 'Profile file not found: ' *)
				T_Visu.ptrT_ExchgParam^.T_Visu.T_Message.sDynamicTextEnglish:=CONCAT(T_Visu.ptrT_ExchgParam^.T_Visu.T_Message.sDynamicTextEnglish,sToLoadProfileName);
				(* For German Language *)
				T_Visu.ptrT_ExchgParam^.T_Visu.T_Message.sDynamicTextDeutsch:=CONCAT(T_ErrorList.asErrorListDeutsch.T_LanguagList[50],sTmpDynamicText);	(* 'Profile file not found: ' *)
				T_Visu.ptrT_ExchgParam^.T_Visu.T_Message.sDynamicTextDeutsch:=CONCAT(T_Visu.ptrT_ExchgParam^.T_Visu.T_Message.sDynamicTextDeutsch,sToLoadProfileName);
				(* For French Language *)
				T_Visu.ptrT_ExchgParam^.T_Visu.T_Message.sDynamicTextFrancais:=CONCAT(T_ErrorList.asErrorListFrancais.T_LanguagList[50],sTmpDynamicText);	(* 'Profile file not found: ' *)
				T_Visu.ptrT_ExchgParam^.T_Visu.T_Message.sDynamicTextFrancais:=CONCAT(T_Visu.ptrT_ExchgParam^.T_Visu.T_Message.sDynamicTextFrancais,sToLoadProfileName);
				T_Visu.ptrT_ExchgParam^.T_SafetyCtrl.xSetForceError:=TRUE;
				T_Visu.ptrT_ExchgParam^.T_SafetyCtrl.diSetForceErrorNr:=1;	(* Datei für Profile nicht gefunden *)
			END_IF;
			xUpdateProfileList:=TRUE;
			T_Visu.T_CtrleAction.xDone:=TRUE;
			T_Visu.T_CtrleAction.xErr:=FALSE;
			T_Visu.T_CtrleAction.udiErrorID:=16#0;
			xAction_CopyProfileToProcess:=FALSE;
		(* not ready *)
		95:	TimerNotReady(IN:=TRUE);
			xAction_CopyProfileToProcess:=FALSE;
		(* Error *)
		99:	T_Visu.T_CtrleAction.xDone:=FALSE;
			T_Visu.T_CtrleAction.xErr:=TRUE;
			T_Visu.T_CtrleAction.udiErrorID:=16#F1000 + T_Profile.T_Ctrle.iFunction;
			xAction_CopyProfileToProcess:=FALSE;
		END_CASE
	END_IF

(* Load profile to process image *)
	IF xAction_LoadProfileToProcessImage THEN
		(* Step import/export profile value *)
		CASE iStepAction OF
		(* Display message to ask for confirmation *)
		1:	T_Visu.ptrT_ExchgParam^.T_Visu.T_Message.iState:=111;
			(* next step *)
			iStepAction:=10;
		(* waiting for key <Enter> or <Esc> *)
		10:	IF RisingEdgeKeyPanel_Enter.Q THEN
				xProfileFileNotFound:=FALSE;
				(* Display message transfering *)
				T_Visu.ptrT_ExchgParam^.T_Visu.T_Message.iState:=15;
				(* next step *)
				iStepAction:=20;
			ELSE
				IF RisingEdgeKeyPanel_Esc.Q THEN iStepAction:=90; END_IF
				(* An other message has been displayed, stop import/export action *)
				IF T_Visu.ptrT_ExchgParam^.T_Visu.T_Message.iState<>105 AND  T_Visu.ptrT_ExchgParam^.T_Visu.T_Message.iState<>111THEN iStepAction:=90; END_IF
			END_IF
		(* Init. reading profile file *)
		20:	IF T_NovRam.T_Data.T_IDProfileStation[T_Visu.ptrT_ExchgParam^.T_ProfileCommon.T_Id.iNumber].sName <> '' THEN
			(* Profile name exists *)
				T_Profile.T_Id.iNumber:=T_Visu.ptrT_ExchgParam^.T_ProfileCommon.T_Id.iNumber;
				T_Profile.T_Id.sName:=T_NovRam.T_Data.T_IDProfileStation[T_Visu.ptrT_ExchgParam^.T_ProfileCommon.T_Id.iNumber].sName;
				T_Profile.T_Ctrle.iFunction:=1;
				T_Profile.T_Ctrle.xExecute:=TRUE;
				(* Display info message *)
				T_Visu.ptrT_ExchgParam^.T_Visu.T_Message.iState:=15;
				(* next step *)
				iStepAction:=30;
			(* Display info message 'file does not exists *)
			ELSE
				T_Visu.ptrT_ExchgParam^.T_Visu.T_Message.iState:=11;
				(* next step *)
				iStepAction:=50;
				xStepActionDone:=FALSE;
				tTimeOutAction:=TimerAction.ET+T#2s;
			END_IF
		(* waiting confirmation signal *)
		30:	IF NOT T_Profile.T_Ctrle.xExecute AND T_Profile.T_Ctrle.xDone THEN
			(* Copy profile to online value *)
				T_NovRam.T_Data.T_ProcessImageData:=T_NovRam.T_Data.T_ProcessImageLoadData;
				xResetParaListValue:=TRUE;
				(* next step *)
				iStepAction:=60;
			END_IF
			IF T_Profile.T_Ctrle.xErr THEN
				IF T_Profile.T_Id.iNumber > 1 THEN
				(* Reset profile value, display message and reset profile error *)
					(*xFctResetProfileValue(ptrProfileData:=ADR(T_Profile.T_DataOnline));*)
					T_Visu.ptrT_ExchgParam^.T_ProfileCommon.T_Id.sName:='';
					(* Profile will be erased from the profile list *)
					T_NovRam.T_Data.T_IDProfileStation[T_Visu.ptrT_ExchgParam^.T_ProfileCommon.T_Id.iNumber].sName:='';
					xUpdateProfileList:=TRUE;
					(* Display info message 'file does not exists *)
					T_Visu.ptrT_ExchgParam^.T_Visu.T_Message.iState:=11;
					(* Reset control profile *)
					T_Profile.T_Ctrle.xReset:=TRUE;
					(* next step *)
					iStepAction:=40;
					xStepActionDone:=FALSE;
					(* use tmp timer to diplay message *)
					TimerONTmp(IN:=FALSE);
					TimerONTmp.PT:=T#1s;
				ELSE
					xProfileFileNotFound:=TRUE;
					iToLoadProfileNr:=1;
					sToLoadProfileName:='Default';
					(* Set Static Default Parameter *)
(*
					IF xFctSetDefaultValueProfileOnlineChange(ptrNovRAM:=ADR(T_WorkingData),
									ptrDefaultProfilStandProcPara:=ADR(T_DefaultProfilStandProcPara),
									bActiveStation:=T_Visu.ptrT_ExchgParam^.T_Visu.bActivStation) THEN
						T_WorkingData.T_Station[T_Visu.ptrT_ExchgParam^.T_Visu.bActivStation].T_StProcess:=T_DefaultProfilStandProcPara[T_Visu.ptrT_ExchgParam^.T_Visu.bActivStation];
						T_ActualProfilStandProcPara[T_Visu.ptrT_ExchgParam^.T_Visu.bActivStation]:=T_DefaultProfilStandProcPara[T_Visu.ptrT_ExchgParam^.T_Visu.bActivStation];
						T_Visu.ptrT_ExchgParam^.T_StationCommon.T_ParamStProcess:=T_DefaultProfilStandProcPara[T_Visu.ptrT_ExchgParam^.T_Visu.bActivStation];
						T_WorkingData.T_Station[T_Visu.ptrT_ExchgParam^.T_Visu.bActivStation].T_InfoProcess.iProfile:=1;
						T_WorkingData.T_Station[T_Visu.ptrT_ExchgParam^.T_Visu.bActivStation].T_Config.iProfile:=1;
						T_WorkingData.T_Station[T_Visu.ptrT_ExchgParam^.T_Visu.bActivStation].T_InfoProcess.sProfileName:='Default';
						T_Visu.ptrT_ExchgParam^.T_StationCommon.T_InfoProcess.iProfile:=1;
						T_Visu.ptrT_ExchgParam^.T_StationCommon.T_InfoProcess.sProfileName:='Default';
						(* Reset control profile *)
						T_Profile.T_Ctrle.xReset:=TRUE;
						(* next step *)
						iStepAction:=60;
					END_IF;
*)
				END_IF;
			END_IF
		(* Wait delay timer *)
		40:	IF TimerONTmp.Q THEN
				T_Visu.ptrT_ExchgParam^.T_Visu.T_Message.iState:=0;
				(* next step *)
				iStepAction:=60;
			END_IF
		(* delay time out *)
		50:	IF TimerAction.Q THEN xAction_LoadProfileToProcessImage:=FALSE; END_IF
		(* active saving data NovRAM *)
		60:	IF NOT(xResetParaListValue) THEN
				xAction_SaveNovRAMWithoutConfirm:=TRUE;
				iStepActionNovRam:=1;
				(* next step *)
				iStepAction:=80;
			END_IF;
		(* waiting confirm saving NovRAM action *)
		80:	IF NOT xAction_SaveNovRAMWithoutConfirm THEN
				iStepAction:=90;
			END_IF;
		(* save done *)
		90:	IF xProfileFileNotFound THEN
				xProfileFileNotFound:=FALSE;
				sTmpDynamicText:=INT_TO_STRING(iToLoadProfileNr);
				sTmpDynamicText:=CONCAT(sTmpDynamicText,' ');
				sTmpDynamicText:=CONCAT(sTmpDynamicText,sToLoadProfileName);
				(* For English Language *)
				T_Visu.ptrT_ExchgParam^.T_Visu.T_Message.sDynamicTextEnglish:=CONCAT(T_ErrorList.asErrorListEnglish.T_LanguagList[50],sTmpDynamicText);	(* 'Profile file not found: ' *)
				T_Visu.ptrT_ExchgParam^.T_Visu.T_Message.sDynamicTextEnglish:=CONCAT(T_Visu.ptrT_ExchgParam^.T_Visu.T_Message.sDynamicTextEnglish,T_ErrorList.asErrorListEnglish.T_LanguagList[51]);	(* ' -->Load static default parameter' *)
				(* For German Language *)
				T_Visu.ptrT_ExchgParam^.T_Visu.T_Message.sDynamicTextDeutsch:=CONCAT(T_ErrorList.asErrorListDeutsch.T_LanguagList[50],sTmpDynamicText);	(* 'Profile file not found: ' *)
				T_Visu.ptrT_ExchgParam^.T_Visu.T_Message.sDynamicTextDeutsch:=CONCAT(T_Visu.ptrT_ExchgParam^.T_Visu.T_Message.sDynamicTextDeutsch,T_ErrorList.asErrorListDeutsch.T_LanguagList[51]);	(* ' -->Load static default parameter' *)
				(* For French Language *)
				T_Visu.ptrT_ExchgParam^.T_Visu.T_Message.sDynamicTextFrancais:=CONCAT(T_ErrorList.asErrorListFrancais.T_LanguagList[50],sTmpDynamicText);	(* 'Profile file not found: ' *)
				T_Visu.ptrT_ExchgParam^.T_Visu.T_Message.sDynamicTextFrancais:=CONCAT(T_Visu.ptrT_ExchgParam^.T_Visu.T_Message.sDynamicTextFrancais,T_ErrorList.asErrorListFrancais.T_LanguagList[51]);	(* ' -->Load static default parameter' *)
				T_Visu.ptrT_ExchgParam^.T_SafetyCtrl.xSetForceError:=TRUE;
				T_Visu.ptrT_ExchgParam^.T_SafetyCtrl.diSetForceErrorNr:=1;	(* Datei für Profile nicht gefunden *)
			END_IF;
			T_Visu.ptrT_ExchgParam^.T_Visu.T_Message.iState:=0;
			T_Visu.T_CtrleAction.xDone:=TRUE;
			T_Visu.T_CtrleAction.xNotReady:=FALSE;
			T_Visu.T_CtrleAction.xErr:=FALSE;
			T_Visu.T_CtrleAction.udiErrorID:=0;
			xAction_LoadProfileToProcessImage:=FALSE;
		(* Action not ready *)
		95:	TimerNotReady(IN:=TRUE);
			xAction_LoadProfileToProcessImage:=FALSE;
		(* error *)
		99:	T_Visu.T_CtrleAction.xDone:=FALSE;
			T_Visu.T_CtrleAction.xNotReady:=FALSE;
			T_Visu.T_CtrleAction.xErr:=TRUE;
			T_Visu.T_CtrleAction.udiErrorID:=16#F1000 + T_Profile.T_Ctrle.iFunction;
			xAction_LoadProfileToProcessImage:=FALSE;
		END_CASE
	END_IF

